LIN {X 261.750,Y 124.846,Z 181.546,A -154.500,B 90.000,C 0.000} C_DIS
LIN {X 261.491,Y 125.389,Z 179.119,A -154.382,B 90.000,C 0.000} C_DIS
LIN {X 261.280,Y 125.829,Z 176.668,A -154.285,B 90.000,C 0.000} C_DIS
LIN {X 261.097,Y 126.208,Z 174.203,A -154.202,B 90.000,C 0.000} C_DIS
LIN {X 261.001,Y 126.406,Z 172.680,A -154.159,B 90.000,C 0.000} C_DIS
LIN {X 260.699,Y 127.028,Z 175.082,A -154.022,B 90.000,C 0.000} C_DIS
LIN {X 260.678,Y 127.070,Z 175.258,A -154.013,B 90.000,C 0.000} C_DIS
LIN {X 260.668,Y 127.091,Z 175.443,A -154.008,B 90.000,C 0.000} C_DIS
LIN {X 260.648,Y 127.131,Z 175.543,A -153.999,B 90.000,C 0.000} C_DIS
LIN {X 260.511,Y 127.412,Z 176.567,A -153.938,B 90.000,C 0.000} C_DIS
LIN {X 260.496,Y 127.443,Z 176.806,A -153.931,B 90.000,C 0.000} C_DIS
LIN {X 260.198,Y 128.050,Z 179.115,A -153.797,B 90.000,C 0.000} C_DIS
LIN {X 260.188,Y 128.071,Z 179.244,A -153.792,B 90.000,C 0.000} C_DIS
LIN {X 260.152,Y 128.145,Z 179.466,A -153.776,B 90.000,C 0.000} C_DIS
LIN {X 260.141,Y 128.166,Z 179.594,A -153.772,B 90.000,C 0.000} C_DIS
LIN {X 259.890,Y 128.674,Z 181.403,A -153.660,B 90.000,C 0.000} C_DIS
LIN {X 259.860,Y 128.735,Z 181.801,A -153.646,B 90.000,C 0.000} C_DIS
LIN {X 259.844,Y 128.768,Z 181.915,A -153.639,B 90.000,C 0.000} C_DIS
LIN {X 259.830,Y 128.797,Z 181.972,A -153.633,B 90.000,C 0.000} C_DIS
LIN {X 259.824,Y 128.808,Z 182.029,A -153.630,B 90.000,C 0.000} C_DIS
LIN {X 259.588,Y 129.283,Z 183.707,A -153.525,B 90.000,C 0.000} C_DIS
LIN {X 259.577,Y 129.304,Z 183.864,A -153.521,B 90.000,C 0.000} C_DIS
LIN {X 259.564,Y 129.330,Z 183.963,A -153.515,B 90.000,C 0.000} C_DIS
LIN {X 259.518,Y 129.423,Z 184.177,A -153.494,B 90.000,C 0.000} C_DIS
LIN {X 259.392,Y 129.675,Z 185.123,A -153.439,B 90.000,C 0.000} C_DIS
LIN {X 259.382,Y 129.696,Z 185.286,A -153.434,B 90.000,C 0.000} C_DIS
LIN {X 259.358,Y 129.744,Z 185.386,A -153.423,B 90.000,C 0.000} C_DIS
LIN {X 259.343,Y 129.773,Z 185.423,A -153.417,B 90.000,C 0.000} C_DIS
LIN {X 259.334,Y 129.792,Z 185.531,A -153.413,B 90.000,C 0.000} C_DIS
LIN {X 259.124,Y 130.210,Z 186.922,A -153.320,B 90.000,C 0.000} C_DIS
LIN {X 258.879,Y 130.697,Z 188.742,A -153.213,B 90.000,C 0.000} C_DIS
LIN {X 258.539,Y 131.368,Z 190.848,A -153.064,B 90.000,C 0.000} C_DIS
LIN {X 258.522,Y 131.401,Z 191.075,A -153.057,B 90.000,C 0.000} C_DIS
LIN {X 258.356,Y 131.727,Z 191.986,A -152.985,B 90.000,C 0.000} C_DIS
LIN {X 258.326,Y 131.787,Z 192.346,A -152.971,B 90.000,C 0.000} C_DIS
LIN {X 258.310,Y 131.819,Z 192.384,A -152.964,B 90.000,C 0.000} C_DIS
LIN {X 258.290,Y 131.857,Z 192.498,A -152.956,B 90.000,C 0.000} C_DIS
LIN {X 258.283,Y 131.871,Z 192.611,A -152.952,B 90.000,C 0.000} C_DIS
LIN {X 258.179,Y 132.075,Z 193.180,A -152.907,B 90.000,C 0.000} C_DIS
LIN {X 258.171,Y 132.089,Z 193.294,A -152.904,B 90.000,C 0.000} C_DIS
LIN {X 258.154,Y 132.122,Z 193.408,A -152.897,B 90.000,C 0.000} C_DIS
LIN {X 258.140,Y 132.150,Z 193.465,A -152.891,B 90.000,C 0.000} C_DIS
LIN {X 258.134,Y 132.162,Z 193.522,A -152.888,B 90.000,C 0.000} C_DIS
LIN {X 257.980,Y 132.463,Z 194.356,A -152.821,B 90.000,C 0.000} C_DIS
LIN {X 257.975,Y 132.473,Z 194.455,A -152.819,B 90.000,C 0.000} C_DIS
LIN {X 257.839,Y 132.737,Z 195.229,A -152.760,B 90.000,C 0.000} C_DIS
LIN {X 257.834,Y 132.747,Z 195.342,A -152.758,B 90.000,C 0.000} C_DIS
LIN {X 257.799,Y 132.815,Z 195.542,A -152.743,B 90.000,C 0.000} C_DIS
LIN {X 257.793,Y 132.826,Z 195.627,A -152.741,B 90.000,C 0.000} C_DIS
LIN {X 257.655,Y 133.093,Z 196.400,A -152.681,B 90.000,C 0.000} C_DIS
LIN {X 257.650,Y 133.103,Z 196.500,A -152.679,B 90.000,C 0.000} C_DIS
LIN {X 257.529,Y 133.337,Z 197.076,A -152.627,B 90.000,C 0.000} C_DIS
LIN {X 257.435,Y 133.518,Z 197.632,A -152.587,B 90.000,C 0.000} C_DIS
LIN {X 257.056,Y 134.247,Z 199.808,A -152.424,B 90.000,C 0.000} C_DIS
LIN {X 256.932,Y 134.483,Z 200.387,A -152.372,B 90.000,C 0.000} C_DIS
LIN {X 256.928,Y 134.491,Z 200.486,A -152.370,B 90.000,C 0.000} C_DIS
LIN {X 256.816,Y 134.705,Z 201.032,A -152.322,B 90.000,C 0.000} C_DIS
LIN {X 256.810,Y 134.716,Z 201.146,A -152.320,B 90.000,C 0.000} C_DIS
LIN {X 256.793,Y 134.749,Z 201.260,A -152.312,B 90.000,C 0.000} C_DIS
LIN {X 256.778,Y 134.777,Z 201.316,A -152.306,B 90.000,C 0.000} C_DIS
LIN {X 256.417,Y 135.464,Z 203.137,A -152.153,B 90.000,C 0.000} C_DIS
LIN {X 256.396,Y 135.504,Z 203.251,A -152.144,B 90.000,C 0.000} C_DIS
LIN {X 256.367,Y 135.557,Z 203.338,A -152.132,B 90.000,C 0.000} C_DIS
LIN {X 256.288,Y 135.707,Z 203.870,A -152.098,B 90.000,C 0.000} C_DIS
LIN {X 256.269,Y 135.744,Z 203.927,A -152.090,B 90.000,C 0.000} C_DIS
LIN {X 256.128,Y 136.010,Z 204.533,A -152.031,B 90.000,C 0.000} C_DIS
LIN {X 256.051,Y 136.154,Z 205.052,A -151.998,B 90.000,C 0.000} C_DIS
LIN {X 256.028,Y 136.196,Z 205.122,A -151.989,B 90.000,C 0.000} C_DIS
LIN {X 255.803,Y 136.620,Z 206.186,A -151.894,B 90.000,C 0.000} C_DIS
LIN {X 255.794,Y 136.635,Z 206.270,A -151.891,B 90.000,C 0.000} C_DIS
LIN {X 255.561,Y 137.072,Z 207.291,A -151.793,B 90.000,C 0.000} C_DIS
LIN {X 255.543,Y 137.106,Z 207.333,A -151.785,B 90.000,C 0.000} C_DIS
LIN {X 255.484,Y 137.214,Z 207.749,A -151.761,B 90.000,C 0.000} C_DIS
LIN {X 255.456,Y 137.267,Z 207.803,A -151.749,B 90.000,C 0.000} C_DIS
LIN {X 255.434,Y 137.308,Z 207.916,A -151.740,B 90.000,C 0.000} C_DIS
LIN {X 255.235,Y 137.678,Z 208.850,A -151.657,B 90.000,C 0.000} C_DIS
LIN {X 255.220,Y 137.705,Z 208.884,A -151.651,B 90.000,C 0.000} C_DIS
LIN {X 255.172,Y 137.794,Z 209.086,A -151.631,B 90.000,C 0.000} C_DIS
LIN {X 254.804,Y 138.474,Z 210.647,A -151.478,B 90.000,C 0.000} C_DIS
LIN {X 254.783,Y 138.513,Z 210.761,A -151.469,B 90.000,C 0.000} C_DIS
LIN {X 254.754,Y 138.566,Z 210.842,A -151.457,B 90.000,C 0.000} C_DIS
LIN {X 254.706,Y 138.653,Z 211.023,A -151.438,B 90.000,C 0.000} C_DIS
LIN {X 254.662,Y 138.735,Z 211.155,A -151.419,B 90.000,C 0.000} C_DIS
LIN {X 254.427,Y 139.165,Z 212.216,A -151.322,B 90.000,C 0.000} C_DIS
LIN {X 254.398,Y 139.218,Z 212.297,A -151.311,B 90.000,C 0.000} C_DIS
LIN {X 254.374,Y 139.262,Z 212.411,A -151.301,B 90.000,C 0.000} C_DIS
LIN {X 254.345,Y 139.315,Z 212.492,A -151.289,B 90.000,C 0.000} C_DIS
LIN {X 254.303,Y 139.391,Z 212.661,A -151.271,B 90.000,C 0.000} C_DIS
LIN {X 254.263,Y 139.465,Z 212.780,A -151.255,B 90.000,C 0.000} C_DIS
LIN {X 254.224,Y 139.536,Z 212.973,A -151.239,B 90.000,C 0.000} C_DIS
LIN {X 254.200,Y 139.579,Z 213.172,A -151.229,B 90.000,C 0.000} C_DIS
LIN {X 253.989,Y 139.963,Z 213.976,A -151.143,B 90.000,C 0.000} C_DIS
LIN {X 253.943,Y 140.047,Z 214.108,A -151.124,B 90.000,C 0.000} C_DIS
LIN {X 253.906,Y 140.112,Z 214.264,A -151.109,B 90.000,C 0.000} C_DIS
LIN {X 253.792,Y 140.320,Z 214.630,A -151.062,B 90.000,C 0.000} C_DIS
LIN {X 253.771,Y 140.359,Z 214.744,A -151.053,B 90.000,C 0.000} C_DIS
LIN {X 253.712,Y 140.464,Z 214.915,A -151.030,B 90.000,C 0.000} C_DIS
LIN {X 253.688,Y 140.508,Z 215.028,A -151.020,B 90.000,C 0.000} C_DIS
LIN {X 253.659,Y 140.561,Z 215.105,A -151.008,B 90.000,C 0.000} C_DIS
LIN {X 253.548,Y 140.760,Z 215.521,A -150.963,B 90.000,C 0.000} C_DIS
LIN {X 253.519,Y 140.812,Z 215.597,A -150.951,B 90.000,C 0.000} C_DIS
LIN {X 253.495,Y 140.856,Z 215.711,A -150.941,B 90.000,C 0.000} C_DIS
LIN {X 253.436,Y 140.961,Z 215.882,A -150.917,B 90.000,C 0.000} C_DIS
LIN {X 253.412,Y 141.005,Z 215.996,A -150.907,B 90.000,C 0.000} C_DIS
LIN {X 253.382,Y 141.058,Z 216.072,A -150.895,B 90.000,C 0.000} C_DIS
LIN {X 253.143,Y 141.487,Z 216.805,A -150.798,B 90.000,C 0.000} C_DIS
LIN {X 252.855,Y 142.002,Z 217.779,A -150.682,B 90.000,C 0.000} C_DIS
LIN {X 252.797,Y 142.105,Z 217.992,A -150.658,B 90.000,C 0.000} C_DIS
LIN {X 252.693,Y 142.289,Z 218.286,A -150.616,B 90.000,C 0.000} C_DIS
LIN {X 252.624,Y 142.412,Z 218.442,A -150.589,B 90.000,C 0.000} C_DIS
LIN {X 252.618,Y 142.423,Z 218.499,A -150.586,B 90.000,C 0.000} C_DIS
LIN {X 252.605,Y 142.445,Z 218.556,A -150.581,B 90.000,C 0.000} C_DIS
LIN {X 252.529,Y 142.581,Z 218.764,A -150.550,B 90.000,C 0.000} C_DIS
LIN {X 252.408,Y 142.795,Z 219.122,A -150.502,B 90.000,C 0.000} C_DIS
LIN {X 252.378,Y 142.847,Z 219.182,A -150.490,B 90.000,C 0.000} C_DIS
LIN {X 252.353,Y 142.891,Z 219.296,A -150.480,B 90.000,C 0.000} C_DIS
LIN {X 252.291,Y 143.001,Z 219.466,A -150.455,B 90.000,C 0.000} C_DIS
LIN {X 252.274,Y 143.031,Z 219.499,A -150.448,B 90.000,C 0.000} C_DIS
LIN {X 251.761,Y 143.932,Z 220.886,A -150.243,B 90.000,C 0.000} C_DIS
LIN {X 251.728,Y 143.990,Z 220.946,A -150.230,B 90.000,C 0.000} C_DIS
LIN {X 251.713,Y 144.017,Z 220.981,A -150.224,B 90.000,C 0.000} C_DIS
LIN {X 251.654,Y 144.119,Z 221.173,A -150.201,B 90.000,C 0.000} C_DIS
LIN {X 250.995,Y 145.264,Z 222.709,A -149.940,B 90.000,C 0.000} C_DIS
LIN {X 250.952,Y 145.338,Z 222.766,A -149.923,B 90.000,C 0.000} C_DIS
LIN {X 250.867,Y 145.485,Z 222.937,A -149.889,B 90.000,C 0.000} C_DIS
LIN {X 250.824,Y 145.559,Z 222.982,A -149.872,B 90.000,C 0.000} C_DIS
LIN {X 250.161,Y 146.696,Z 224.246,A -149.612,B 90.000,C 0.000} C_DIS
LIN {X 249.905,Y 147.131,Z 224.706,A -149.513,B 90.000,C 0.000} C_DIS
LIN {X 249.753,Y 147.388,Z 224.928,A -149.454,B 90.000,C 0.000} C_DIS
LIN {X 248.658,Y 149.229,Z 226.216,A -149.030,B 90.000,C 0.000} C_DIS
LIN {X 248.413,Y 149.636,Z 226.445,A -148.937,B 90.000,C 0.000} C_DIS
LIN {X 248.308,Y 149.810,Z 226.460,A -148.897,B 90.000,C 0.000} C_DIS
LIN {X 248.170,Y 150.038,Z 226.328,A -148.844,B 90.000,C 0.000} C_DIS
LIN {X 247.772,Y 150.695,Z 225.771,A -148.692,B 90.000,C 0.000} C_DIS
LIN {X 247.484,Y 151.167,Z 225.386,A -148.583,B 90.000,C 0.000} C_DIS
LIN {X 247.345,Y 151.395,Z 225.255,A -148.530,B 90.000,C 0.000} C_DIS
LIN {X 247.299,Y 151.470,Z 225.156,A -148.513,B 90.000,C 0.000} C_DIS
LIN {X 246.570,Y 152.654,Z 224.116,A -148.238,B 90.000,C 0.000} C_DIS
LIN {X 246.521,Y 152.734,Z 224.018,A -148.219,B 90.000,C 0.000} C_DIS
LIN {X 246.069,Y 153.460,Z 223.362,A -148.051,B 90.000,C 0.000} C_DIS
LIN {X 245.953,Y 153.646,Z 223.134,A -148.007,B 90.000,C 0.000} C_DIS
LIN {X 244.939,Y 155.258,Z 221.514,A -147.631,B 90.000,C 0.000} C_DIS
LIN {X 244.768,Y 155.527,Z 221.240,A -147.568,B 90.000,C 0.000} C_DIS
LIN {X 244.507,Y 155.937,Z 220.768,A -147.472,B 90.000,C 0.000} C_DIS
LIN {X 244.472,Y 155.992,Z 220.682,A -147.459,B 90.000,C 0.000} C_DIS
LIN {X 244.123,Y 156.537,Z 220.149,A -147.331,B 90.000,C 0.000} C_DIS
LIN {X 244.079,Y 156.606,Z 220.034,A -147.315,B 90.000,C 0.000} C_DIS
LIN {X 243.939,Y 156.824,Z 219.782,A -147.264,B 90.000,C 0.000} C_DIS
LIN {X 243.910,Y 156.869,Z 219.759,A -147.253,B 90.000,C 0.000} C_DIS
LIN {X 243.416,Y 157.634,Z 218.840,A -147.073,B 90.000,C 0.000} C_DIS
LIN {X 243.386,Y 157.681,Z 218.755,A -147.062,B 90.000,C 0.000} C_DIS
LIN {X 243.293,Y 157.825,Z 218.583,A -147.028,B 90.000,C 0.000} C_DIS
LIN {X 243.200,Y 157.968,Z 218.351,A -146.995,B 90.000,C 0.000} C_DIS
LIN {X 243.107,Y 158.111,Z 218.186,A -146.961,B 90.000,C 0.000} C_DIS
LIN {X 242.920,Y 158.397,Z 217.804,A -146.894,B 90.000,C 0.000} C_DIS
LIN {X 242.889,Y 158.445,Z 217.788,A -146.882,B 90.000,C 0.000} C_DIS
LIN {X 242.858,Y 158.492,Z 217.763,A -146.871,B 90.000,C 0.000} C_DIS
LIN {X 242.392,Y 159.204,Z 216.749,A -146.703,B 90.000,C 0.000} C_DIS
LIN {X 242.344,Y 159.278,Z 216.678,A -146.686,B 90.000,C 0.000} C_DIS
LIN {X 242.297,Y 159.349,Z 216.591,A -146.669,B 90.000,C 0.000} C_DIS
LIN {X 242.250,Y 159.420,Z 216.471,A -146.652,B 90.000,C 0.000} C_DIS
LIN {X 242.203,Y 159.492,Z 216.388,A -146.635,B 90.000,C 0.000} C_DIS
LIN {X 242.148,Y 159.575,Z 216.229,A -146.615,B 90.000,C 0.000} C_DIS
LIN {X 241.701,Y 160.251,Z 215.249,A -146.455,B 90.000,C 0.000} C_DIS
LIN {X 241.639,Y 160.346,Z 215.211,A -146.433,B 90.000,C 0.000} C_DIS
LIN {X 241.513,Y 160.536,Z 214.821,A -146.388,B 90.000,C 0.000} C_DIS
LIN {X 241.418,Y 160.678,Z 214.665,A -146.354,B 90.000,C 0.000} C_DIS
LIN {X 241.323,Y 160.820,Z 214.461,A -146.320,B 90.000,C 0.000} C_DIS
LIN {X 241.136,Y 161.101,Z 213.937,A -146.253,B 90.000,C 0.000} C_DIS
LIN {X 242.353,Y 159.265,Z 212.755,A -146.689,B 90.000,C 0.000} C_DIS
LIN {X 243.523,Y 157.470,Z 211.467,A -147.112,B 90.000,C 0.000} C_DIS
LIN {X 244.293,Y 156.271,Z 210.534,A -147.393,B 90.000,C 0.000} C_DIS
LIN {X 245.035,Y 155.106,Z 209.566,A -147.666,B 90.000,C 0.000} C_DIS
LIN {X 245.147,Y 154.928,Z 209.396,A -147.708,B 90.000,C 0.000} C_DIS
LIN {X 245.353,Y 154.603,Z 209.168,A -147.784,B 90.000,C 0.000} C_DIS
LIN {X 245.362,Y 154.588,Z 209.113,A -147.787,B 90.000,C 0.000} C_DIS
LIN {X 245.421,Y 154.495,Z 209.021,A -147.809,B 90.000,C 0.000} C_DIS
LIN {X 245.498,Y 154.372,Z 208.933,A -147.838,B 90.000,C 0.000} C_DIS
LIN {X 245.548,Y 154.292,Z 208.843,A -147.857,B 90.000,C 0.000} C_DIS
LIN {X 245.868,Y 153.781,Z 208.428,A -147.976,B 90.000,C 0.000} C_DIS
LIN {X 245.876,Y 153.770,Z 208.372,A -147.978,B 90.000,C 0.000} C_DIS
LIN {X 245.905,Y 153.723,Z 208.315,A -147.989,B 90.000,C 0.000} C_DIS
LIN {X 246.345,Y 153.017,Z 207.660,A -148.153,B 90.000,C 0.000} C_DIS
LIN {X 246.421,Y 152.894,Z 207.575,A -148.182,B 90.000,C 0.000} C_DIS
LIN {X 246.750,Y 152.363,Z 207.063,A -148.305,B 90.000,C 0.000} C_DIS
LIN {X 246.791,Y 152.296,Z 206.978,A -148.321,B 90.000,C 0.000} C_DIS
LIN {X 246.820,Y 152.250,Z 206.892,A -148.332,B 90.000,C 0.000} C_DIS
LIN {X 247.039,Y 151.894,Z 206.586,A -148.414,B 90.000,C 0.000} C_DIS
LIN {X 247.052,Y 151.872,Z 206.551,A -148.419,B 90.000,C 0.000} C_DIS
LIN {X 247.541,Y 151.074,Z 205.811,A -148.604,B 90.000,C 0.000} C_DIS
LIN {X 247.561,Y 151.041,Z 205.697,A -148.612,B 90.000,C 0.000} C_DIS
LIN {X 247.837,Y 150.588,Z 205.299,A -148.717,B 90.000,C 0.000} C_DIS
LIN {X 247.846,Y 150.573,Z 205.242,A -148.720,B 90.000,C 0.000} C_DIS
LIN {X 247.868,Y 150.537,Z 205.185,A -148.728,B 90.000,C 0.000} C_DIS
LIN {X 248.834,Y 148.936,Z 203.527,A -149.098,B 90.000,C 0.000} C_DIS
LIN {X 248.863,Y 148.886,Z 203.478,A -149.109,B 90.000,C 0.000} C_DIS
LIN {X 248.888,Y 148.844,Z 203.365,A -149.119,B 90.000,C 0.000} C_DIS
LIN {X 249.802,Y 147.305,Z 201.620,A -149.473,B 90.000,C 0.000} C_DIS
LIN {X 250.670,Y 145.824,Z 199.802,A -149.812,B 90.000,C 0.000} C_DIS
LIN {X 250.709,Y 145.756,Z 199.719,A -149.827,B 90.000,C 0.000} C_DIS
LIN {X 250.795,Y 145.608,Z 199.609,A -149.861,B 90.000,C 0.000} C_DIS
LIN {X 251.434,Y 144.502,Z 198.183,A -150.114,B 90.000,C 0.000} C_DIS
LIN {X 251.448,Y 144.478,Z 198.130,A -150.119,B 90.000,C 0.000} C_DIS
LIN {X 251.478,Y 144.426,Z 198.045,A -150.131,B 90.000,C 0.000} C_DIS
LIN {X 251.521,Y 144.352,Z 197.960,A -150.148,B 90.000,C 0.000} C_DIS
LIN {X 251.563,Y 144.278,Z 197.895,A -150.165,B 90.000,C 0.000} C_DIS
LIN {X 251.761,Y 143.932,Z 197.394,A -150.243,B 90.000,C 0.000} C_DIS
LIN {X 251.803,Y 143.858,Z 197.334,A -150.260,B 90.000,C 0.000} C_DIS
LIN {X 251.846,Y 143.784,Z 197.248,A -150.277,B 90.000,C 0.000} C_DIS
LIN {X 251.875,Y 143.732,Z 197.163,A -150.289,B 90.000,C 0.000} C_DIS
LIN {X 251.889,Y 143.708,Z 197.110,A -150.294,B 90.000,C 0.000} C_DIS
LIN {X 251.932,Y 143.633,Z 197.020,A -150.311,B 90.000,C 0.000} C_DIS
LIN {X 251.976,Y 143.555,Z 196.952,A -150.329,B 90.000,C 0.000} C_DIS
LIN {X 252.193,Y 143.174,Z 196.348,A -150.416,B 90.000,C 0.000} C_DIS
LIN {X 252.238,Y 143.095,Z 196.282,A -150.434,B 90.000,C 0.000} C_DIS
LIN {X 252.280,Y 143.020,Z 196.192,A -150.451,B 90.000,C 0.000} C_DIS
LIN {X 252.294,Y 142.995,Z 196.139,A -150.456,B 90.000,C 0.000} C_DIS
LIN {X 252.324,Y 142.943,Z 196.054,A -150.468,B 90.000,C 0.000} C_DIS
LIN {X 252.366,Y 142.869,Z 195.968,A -150.485,B 90.000,C 0.000} C_DIS
LIN {X 252.408,Y 142.795,Z 195.907,A -150.502,B 90.000,C 0.000} C_DIS
LIN {X 252.833,Y 142.040,Z 194.805,A -150.673,B 90.000,C 0.000} C_DIS
LIN {X 252.883,Y 141.952,Z 194.714,A -150.693,B 90.000,C 0.000} C_DIS
LIN {X 253.244,Y 141.306,Z 193.754,A -150.839,B 90.000,C 0.000} C_DIS
LIN {X 253.292,Y 141.221,Z 193.658,A -150.859,B 90.000,C 0.000} C_DIS
LIN {X 253.336,Y 141.141,Z 193.501,A -150.877,B 90.000,C 0.000} C_DIS
LIN {X 253.796,Y 140.312,Z 192.272,A -151.064,B 90.000,C 0.000} C_DIS
LIN {X 253.845,Y 140.223,Z 192.182,A -151.084,B 90.000,C 0.000} C_DIS
LIN {X 254.455,Y 139.113,Z 190.433,A -151.334,B 90.000,C 0.000} C_DIS
LIN {X 255.150,Y 137.834,Z 188.401,A -151.622,B 90.000,C 0.000} C_DIS
LIN {X 255.460,Y 137.260,Z 187.428,A -151.751,B 90.000,C 0.000} C_DIS
LIN {X 255.560,Y 137.074,Z 187.135,A -151.792,B 90.000,C 0.000} C_DIS
LIN {X 255.626,Y 136.950,Z 186.979,A -151.820,B 90.000,C 0.000} C_DIS
LIN {X 255.641,Y 136.922,Z 186.865,A -151.826,B 90.000,C 0.000} C_DIS
LIN {X 255.798,Y 136.628,Z 186.373,A -151.892,B 90.000,C 0.000} C_DIS
LIN {X 256.050,Y 136.157,Z 185.556,A -151.998,B 90.000,C 0.000} C_DIS
LIN {X 256.073,Y 136.113,Z 185.442,A -152.008,B 90.000,C 0.000} C_DIS
LIN {X 256.129,Y 136.007,Z 185.272,A -152.031,B 90.000,C 0.000} C_DIS
LIN {X 256.153,Y 135.962,Z 185.158,A -152.041,B 90.000,C 0.000} C_DIS
LIN {X 256.181,Y 135.909,Z 185.081,A -152.053,B 90.000,C 0.000} C_DIS
LIN {X 256.477,Y 135.350,Z 184.134,A -152.178,B 90.000,C 0.000} C_DIS
LIN {X 256.561,Y 135.191,Z 183.770,A -152.214,B 90.000,C 0.000} C_DIS
LIN {X 256.606,Y 135.104,Z 183.654,A -152.233,B 90.000,C 0.000} C_DIS
LIN {X 256.697,Y 134.931,Z 183.292,A -152.272,B 90.000,C 0.000} C_DIS
LIN {X 256.806,Y 134.725,Z 182.917,A -152.318,B 90.000,C 0.000} C_DIS
LIN {X 256.843,Y 134.654,Z 182.813,A -152.334,B 90.000,C 0.000} C_DIS
LIN {X 256.928,Y 134.492,Z 182.484,A -152.370,B 90.000,C 0.000} C_DIS
LIN {X 256.950,Y 134.449,Z 182.423,A -152.379,B 90.000,C 0.000} C_DIS
LIN {X 257.266,Y 133.844,Z 181.127,A -152.514,B 90.000,C 0.000} C_DIS
LIN {X 257.333,Y 133.715,Z 180.936,A -152.543,B 90.000,C 0.000} C_DIS
LIN {X 257.423,Y 133.541,Z 180.574,A -152.581,B 90.000,C 0.000} C_DIS
LIN {X 257.451,Y 133.488,Z 180.493,A -152.593,B 90.000,C 0.000} C_DIS
LIN {X 257.474,Y 133.443,Z 180.379,A -152.603,B 90.000,C 0.000} C_DIS
LIN {X 257.502,Y 133.390,Z 180.302,A -152.615,B 90.000,C 0.000} C_DIS
LIN {X 257.606,Y 133.188,Z 179.886,A -152.660,B 90.000,C 0.000} C_DIS
LIN {X 257.634,Y 133.134,Z 179.810,A -152.672,B 90.000,C 0.000} C_DIS
LIN {X 257.647,Y 133.109,Z 179.758,A -152.678,B 90.000,C 0.000} C_DIS
LIN {X 257.652,Y 133.099,Z 179.687,A -152.680,B 90.000,C 0.000} C_DIS
LIN {X 257.848,Y 132.720,Z 178.966,A -152.764,B 90.000,C 0.000} C_DIS
LIN {X 257.932,Y 132.556,Z 178.501,A -152.801,B 90.000,C 0.000} C_DIS
LIN {X 257.997,Y 132.429,Z 178.241,A -152.829,B 90.000,C 0.000} C_DIS
LIN {X 258.025,Y 132.375,Z 178.160,A -152.841,B 90.000,C 0.000} C_DIS
LIN {X 258.048,Y 132.331,Z 178.046,A -152.851,B 90.000,C 0.000} C_DIS
LIN {X 258.075,Y 132.277,Z 177.965,A -152.862,B 90.000,C 0.000} C_DIS
LIN {X 258.386,Y 131.669,Z 176.591,A -152.997,B 90.000,C 0.000} C_DIS
LIN {X 258.413,Y 131.615,Z 176.510,A -153.009,B 90.000,C 0.000} C_DIS
LIN {X 258.433,Y 131.577,Z 176.396,A -153.018,B 90.000,C 0.000} C_DIS
LIN {X 258.911,Y 130.633,Z 174.131,A -153.227,B 90.000,C 0.000} C_DIS
LIN {X 258.969,Y 130.518,Z 173.878,A -153.252,B 90.000,C 0.000} C_DIS
LIN {X 259.259,Y 129.942,Z 172.129,A -153.380,B 90.000,C 0.000} C_DIS
LIN {X 259.266,Y 129.928,Z 172.015,A -153.383,B 90.000,C 0.000} C_DIS
LIN {X 259.353,Y 129.754,Z 171.389,A -153.421,B 90.000,C 0.000} C_DIS
LIN {X 259.360,Y 129.740,Z 171.275,A -153.424,B 90.000,C 0.000} C_DIS
LIN {X 259.393,Y 129.674,Z 171.119,A -153.439,B 90.000,C 0.000} C_DIS
LIN {X 259.671,Y 129.116,Z 168.698,A -153.562,B 90.000,C 0.000} C_DIS
LIN {X 259.684,Y 129.090,Z 168.587,A -153.568,B 90.000,C 0.000} C_DIS
LIN {X 259.716,Y 129.025,Z 168.431,A -153.582,B 90.000,C 0.000} C_DIS
LIN {X 259.723,Y 129.011,Z 168.317,A -153.585,B 90.000,C 0.000} C_DIS
LIN {X 259.842,Y 128.773,Z 167.322,A -153.638,B 90.000,C 0.000} C_DIS
LIN {X 259.854,Y 128.748,Z 167.232,A -153.643,B 90.000,C 0.000} C_DIS
LIN {X 259.890,Y 128.674,Z 167.079,A -153.660,B 90.000,C 0.000} C_DIS
LIN {X 259.901,Y 128.653,Z 166.894,A -153.664,B 90.000,C 0.000} C_DIS
LIN {X 260.187,Y 128.072,Z 164.480,A -153.792,B 90.000,C 0.000} C_DIS
LIN {X 260.196,Y 128.054,Z 164.405,A -153.796,B 90.000,C 0.000} C_DIS
LIN {X 258.402,Y 127.171,Z 164.405,A -153.796,B 90.000,C 0.000} C_DIS
WAIT SEC 0.1
RET=EKI_SetBool("oxy","torchState",FALSE)
RET = EKI_Send("oxy","torchState")
LIN {X 242.252,Y 119.223,Z 164.405,A -153.796,B 90.000,C 0.000} C_DIS
LIN {X 245.422,Y 112.552,Z 164.348,A -155.364,B 90.000,C 0.000} C_DIS
LIN {X 261.784,Y 120.055,Z 164.348,A -155.364,B 90.000,C 0.000} C_DIS
LIN {X 263.602,Y 120.889,Z 164.348,A -155.364,B 90.000,C 0.000} C_DIS
WAIT SEC 1
RET=EKI_SetBool("oxy","torchState",TRUE)
RET = EKI_Send("oxy","torchState")
LIN {X 263.563,Y 120.973,Z 165.813,A -155.345,B 90.000,C 0.000} C_DIS
LIN {X 263.565,Y 120.969,Z 166.657,A -155.346,B 90.000,C 0.000} C_DIS
LIN {X 263.556,Y 120.989,Z 166.730,A -155.342,B 90.000,C 0.000} C_DIS
LIN {X 263.645,Y 120.795,Z 169.220,A -155.384,B 90.000,C 0.000} C_DIS
LIN {X 263.775,Y 120.510,Z 170.942,A -155.446,B 90.000,C 0.000} C_DIS
LIN {X 264.136,Y 119.717,Z 173.285,A -155.618,B 90.000,C 0.000} C_DIS
LIN {X 264.561,Y 118.775,Z 175.562,A -155.822,B 90.000,C 0.000} C_DIS
LIN {X 264.902,Y 118.011,Z 177.202,A -155.988,B 90.000,C 0.000} C_DIS
LIN {X 265.110,Y 117.545,Z 178.103,A -156.088,B 90.000,C 0.000} C_DIS
LIN {X 265.524,Y 116.607,Z 179.841,A -156.291,B 90.000,C 0.000} C_DIS
LIN {X 265.592,Y 116.450,Z 180.055,A -156.325,B 90.000,C 0.000} C_DIS
LIN {X 265.684,Y 116.242,Z 180.473,A -156.370,B 90.000,C 0.000} C_DIS
LIN {X 265.834,Y 115.897,Z 180.982,A -156.444,B 90.000,C 0.000} C_DIS
LIN {X 265.886,Y 115.778,Z 181.234,A -156.470,B 90.000,C 0.000} C_DIS
LIN {X 266.457,Y 114.457,Z 183.278,A -156.754,B 90.000,C 0.000} C_DIS
LIN {X 266.607,Y 114.108,Z 183.792,A -156.829,B 90.000,C 0.000} C_DIS
LIN {X 266.783,Y 113.695,Z 184.351,A -156.918,B 90.000,C 0.000} C_DIS
LIN {X 266.811,Y 113.630,Z 184.483,A -156.932,B 90.000,C 0.000} C_DIS
LIN {X 266.856,Y 113.525,Z 184.520,A -156.954,B 90.000,C 0.000} C_DIS
LIN {X 266.945,Y 113.316,Z 184.911,A -156.999,B 90.000,C 0.000} C_DIS
LIN {X 267.011,Y 113.159,Z 185.073,A -157.033,B 90.000,C 0.000} C_DIS
LIN {X 267.034,Y 113.105,Z 185.158,A -157.045,B 90.000,C 0.000} C_DIS
LIN {X 267.071,Y 113.017,Z 185.253,A -157.063,B 90.000,C 0.000} C_DIS
LIN {X 267.121,Y 112.901,Z 185.449,A -157.088,B 90.000,C 0.000} C_DIS
LIN {X 267.564,Y 111.845,Z 186.835,A -157.314,B 90.000,C 0.000} C_DIS
LIN {X 267.695,Y 111.533,Z 187.250,A -157.381,B 90.000,C 0.000} C_DIS
LIN {X 267.717,Y 111.480,Z 187.292,A -157.393,B 90.000,C 0.000} C_DIS
LIN {X 267.738,Y 111.428,Z 187.309,A -157.404,B 90.000,C 0.000} C_DIS
LIN {X 267.891,Y 111.060,Z 187.840,A -157.483,B 90.000,C 0.000} C_DIS
LIN {X 267.935,Y 110.955,Z 187.882,A -157.505,B 90.000,C 0.000} C_DIS
LIN {X 268.087,Y 110.587,Z 188.412,A -157.584,B 90.000,C 0.000} C_DIS
LIN {X 268.109,Y 110.534,Z 188.430,A -157.595,B 90.000,C 0.000} C_DIS
LIN {X 268.130,Y 110.481,Z 188.454,A -157.606,B 90.000,C 0.000} C_DIS
LIN {X 268.583,Y 109.376,Z 189.820,A -157.842,B 90.000,C 0.000} C_DIS
LIN {X 268.603,Y 109.327,Z 189.854,A -157.853,B 90.000,C 0.000} C_DIS
LIN {X 268.637,Y 109.243,Z 189.941,A -157.871,B 90.000,C 0.000} C_DIS
LIN {X 268.661,Y 109.185,Z 190.035,A -157.883,B 90.000,C 0.000} C_DIS
LIN {X 269.243,Y 107.740,Z 191.588,A -158.191,B 90.000,C 0.000} C_DIS
LIN {X 269.266,Y 107.684,Z 191.613,A -158.203,B 90.000,C 0.000} C_DIS
LIN {X 269.300,Y 107.599,Z 191.695,A -158.221,B 90.000,C 0.000} C_DIS
LIN {X 269.328,Y 107.528,Z 191.786,A -158.236,B 90.000,C 0.000} C_DIS
LIN {X 269.357,Y 107.455,Z 191.847,A -158.251,B 90.000,C 0.000} C_DIS
LIN {X 269.412,Y 107.317,Z 191.934,A -158.281,B 90.000,C 0.000} C_DIS
LIN {X 269.566,Y 106.932,Z 192.348,A -158.363,B 90.000,C 0.000} C_DIS
LIN {X 269.620,Y 106.793,Z 192.554,A -158.392,B 90.000,C 0.000} C_DIS
LIN {X 269.842,Y 106.233,Z 193.043,A -158.511,B 90.000,C 0.000} C_DIS
LIN {X 269.894,Y 106.101,Z 193.255,A -158.539,B 90.000,C 0.000} C_DIS
LIN {X 270.373,Y 104.874,Z 194.375,A -158.799,B 90.000,C 0.000} C_DIS
LIN {X 270.390,Y 104.829,Z 194.435,A -158.809,B 90.000,C 0.000} C_DIS
LIN {X 270.409,Y 104.779,Z 194.463,A -158.819,B 90.000,C 0.000} C_DIS
LIN {X 270.442,Y 104.695,Z 194.549,A -158.837,B 90.000,C 0.000} C_DIS
LIN {X 270.467,Y 104.632,Z 194.638,A -158.851,B 90.000,C 0.000} C_DIS
LIN {X 270.535,Y 104.454,Z 194.762,A -158.888,B 90.000,C 0.000} C_DIS
LIN {X 270.745,Y 103.910,Z 195.249,A -159.004,B 90.000,C 0.000} C_DIS
LIN {X 270.769,Y 103.848,Z 195.339,A -159.017,B 90.000,C 0.000} C_DIS
LIN {X 270.801,Y 103.763,Z 195.425,A -159.035,B 90.000,C 0.000} C_DIS
LIN {X 270.820,Y 103.714,Z 195.453,A -159.045,B 90.000,C 0.000} C_DIS
LIN {X 270.840,Y 103.661,Z 195.513,A -159.056,B 90.000,C 0.000} C_DIS
LIN {X 271.527,Y 101.849,Z 197.093,A -159.439,B 90.000,C 0.000} C_DIS
LIN {X 271.664,Y 101.483,Z 197.391,A -159.516,B 90.000,C 0.000} C_DIS
LIN {X 271.685,Y 101.425,Z 197.451,A -159.528,B 90.000,C 0.000} C_DIS
LIN {X 271.704,Y 101.376,Z 197.479,A -159.539,B 90.000,C 0.000} C_DIS
LIN {X 271.766,Y 101.208,Z 197.644,A -159.574,B 90.000,C 0.000} C_DIS
LIN {X 271.785,Y 101.159,Z 197.663,A -159.585,B 90.000,C 0.000} C_DIS
LIN {X 272.177,Y 100.099,Z 198.529,A -159.808,B 90.000,C 0.000} C_DIS
LIN {X 272.199,Y 100.038,Z 198.595,A -159.821,B 90.000,C 0.000} C_DIS
LIN {X 272.212,Y 100.003,Z 198.624,A -159.828,B 90.000,C 0.000} C_DIS
LIN {X 272.335,Y 99.667,Z 198.870,A -159.899,B 90.000,C 0.000} C_DIS
LIN {X 272.356,Y 99.611,Z 198.936,A -159.911,B 90.000,C 0.000} C_DIS
LIN {X 272.369,Y 99.576,Z 198.966,A -159.918,B 90.000,C 0.000} C_DIS
LIN {X 273.063,Y 97.656,Z 200.406,A -160.321,B 90.000,C 0.000} C_DIS
LIN {X 273.091,Y 97.578,Z 200.466,A -160.338,B 90.000,C 0.000} C_DIS
LIN {X 273.129,Y 97.470,Z 200.517,A -160.360,B 90.000,C 0.000} C_DIS
LIN {X 273.149,Y 97.414,Z 200.577,A -160.372,B 90.000,C 0.000} C_DIS
LIN {X 273.269,Y 97.076,Z 200.822,A -160.443,B 90.000,C 0.000} C_DIS
LIN {X 273.339,Y 96.881,Z 200.978,A -160.484,B 90.000,C 0.000} C_DIS
LIN {X 273.358,Y 96.827,Z 201.004,A -160.495,B 90.000,C 0.000} C_DIS
LIN {X 273.377,Y 96.773,Z 201.018,A -160.506,B 90.000,C 0.000} C_DIS
LIN {X 273.528,Y 96.344,Z 201.376,A -160.596,B 90.000,C 0.000} C_DIS
LIN {X 273.665,Y 95.955,Z 201.633,A -160.678,B 90.000,C 0.000} C_DIS
LIN {X 273.717,Y 95.807,Z 201.713,A -160.709,B 90.000,C 0.000} C_DIS
LIN {X 273.904,Y 95.270,Z 202.118,A -160.821,B 90.000,C 0.000} C_DIS
LIN {X 273.932,Y 95.190,Z 202.170,A -160.838,B 90.000,C 0.000} C_DIS
LIN {X 273.972,Y 95.076,Z 202.268,A -160.862,B 90.000,C 0.000} C_DIS
LIN {X 274.091,Y 94.733,Z 202.447,A -160.934,B 90.000,C 0.000} C_DIS
LIN {X 274.133,Y 94.612,Z 202.544,A -160.959,B 90.000,C 0.000} C_DIS
LIN {X 274.818,Y 92.601,Z 203.862,A -161.379,B 90.000,C 0.000} C_DIS
LIN {X 274.942,Y 92.234,Z 204.078,A -161.455,B 90.000,C 0.000} C_DIS
LIN {X 274.979,Y 92.122,Z 204.162,A -161.478,B 90.000,C 0.000} C_DIS
LIN {X 275.097,Y 91.770,Z 204.305,A -161.552,B 90.000,C 0.000} C_DIS
LIN {X 275.134,Y 91.660,Z 204.391,A -161.575,B 90.000,C 0.000} C_DIS
LIN {X 275.205,Y 91.446,Z 204.495,A -161.619,B 90.000,C 0.000} C_DIS
LIN {X 275.625,Y 90.172,Z 205.242,A -161.884,B 90.000,C 0.000} C_DIS
LIN {X 275.650,Y 90.095,Z 205.303,A -161.900,B 90.000,C 0.000} C_DIS
LIN {X 275.668,Y 90.041,Z 205.328,A -161.912,B 90.000,C 0.000} C_DIS
LIN {X 275.685,Y 89.987,Z 205.341,A -161.923,B 90.000,C 0.000} C_DIS
LIN {X 275.824,Y 89.560,Z 205.531,A -162.011,B 90.000,C 0.000} C_DIS
LIN {X 276.068,Y 88.805,Z 205.996,A -162.168,B 90.000,C 0.000} C_DIS
LIN {X 276.090,Y 88.737,Z 206.007,A -162.182,B 90.000,C 0.000} C_DIS
LIN {X 276.262,Y 88.200,Z 206.259,A -162.294,B 90.000,C 0.000} C_DIS
LIN {X 276.555,Y 87.278,Z 206.726,A -162.485,B 90.000,C 0.000} C_DIS
LIN {X 276.593,Y 87.156,Z 206.747,A -162.510,B 90.000,C 0.000} C_DIS
LIN {X 276.623,Y 87.061,Z 206.774,A -162.530,B 90.000,C 0.000} C_DIS
LIN {X 276.787,Y 86.540,Z 207.016,A -162.638,B 90.000,C 0.000} C_DIS
LIN {X 276.816,Y 86.445,Z 207.025,A -162.657,B 90.000,C 0.000} C_DIS
LIN {X 277.064,Y 85.649,Z 207.363,A -162.822,B 90.000,C 0.000} C_DIS
LIN {X 277.080,Y 85.594,Z 207.376,A -162.833,B 90.000,C 0.000} C_DIS
LIN {X 277.127,Y 85.445,Z 207.452,A -162.864,B 90.000,C 0.000} C_DIS
LIN {X 277.178,Y 85.278,Z 207.483,A -162.899,B 90.000,C 0.000} C_DIS
LIN {X 277.229,Y 85.111,Z 207.423,A -162.933,B 90.000,C 0.000} C_DIS
LIN {X 277.265,Y 84.996,Z 207.256,A -162.957,B 90.000,C 0.000} C_DIS
LIN {X 277.464,Y 84.343,Z 205.986,A -163.092,B 90.000,C 0.000} C_DIS
LIN {X 277.480,Y 84.290,Z 205.925,A -163.103,B 90.000,C 0.000} C_DIS
LIN {X 277.533,Y 84.116,Z 205.641,A -163.139,B 90.000,C 0.000} C_DIS
LIN {X 277.546,Y 84.074,Z 205.527,A -163.147,B 90.000,C 0.000} C_DIS
LIN {X 277.563,Y 84.017,Z 205.438,A -163.159,B 90.000,C 0.000} C_DIS
LIN {X 277.650,Y 83.730,Z 204.853,A -163.218,B 90.000,C 0.000} C_DIS
LIN {X 277.653,Y 83.720,Z 204.782,A -163.221,B 90.000,C 0.000} C_DIS
LIN {X 277.661,Y 83.693,Z 204.730,A -163.226,B 90.000,C 0.000} C_DIS
LIN {X 277.678,Y 83.635,Z 204.649,A -163.238,B 90.000,C 0.000} C_DIS
LIN {X 277.699,Y 83.567,Z 204.490,A -163.252,B 90.000,C 0.000} C_DIS
LIN {X 277.890,Y 82.930,Z 203.163,A -163.383,B 90.000,C 0.000} C_DIS
LIN {X 277.914,Y 82.847,Z 203.046,A -163.401,B 90.000,C 0.000} C_DIS
LIN {X 277.939,Y 82.763,Z 202.877,A -163.418,B 90.000,C 0.000} C_DIS
LIN {X 277.956,Y 82.705,Z 202.796,A -163.430,B 90.000,C 0.000} C_DIS
LIN {X 277.971,Y 82.657,Z 202.682,A -163.440,B 90.000,C 0.000} C_DIS
LIN {X 278.004,Y 82.545,Z 202.511,A -163.463,B 90.000,C 0.000} C_DIS
LIN {X 278.018,Y 82.500,Z 202.469,A -163.472,B 90.000,C 0.000} C_DIS
LIN {X 278.309,Y 81.512,Z 200.191,A -163.675,B 90.000,C 0.000} C_DIS
LIN {X 278.345,Y 81.390,Z 199.951,A -163.701,B 90.000,C 0.000} C_DIS
LIN {X 278.354,Y 81.359,Z 199.837,A -163.707,B 90.000,C 0.000} C_DIS
LIN {X 278.491,Y 80.886,Z 198.861,A -163.804,B 90.000,C 0.000} C_DIS
LIN {X 278.502,Y 80.851,Z 198.642,A -163.812,B 90.000,C 0.000} C_DIS
LIN {X 278.517,Y 80.798,Z 198.561,A -163.822,B 90.000,C 0.000} C_DIS
LIN {X 278.556,Y 80.664,Z 198.301,A -163.850,B 90.000,C 0.000} C_DIS
LIN {X 278.560,Y 80.651,Z 198.230,A -163.853,B 90.000,C 0.000} C_DIS
LIN {X 278.770,Y 79.921,Z 196.480,A -164.003,B 90.000,C 0.000} C_DIS
LIN {X 278.784,Y 79.873,Z 196.253,A -164.013,B 90.000,C 0.000} C_DIS
LIN {X 278.942,Y 79.317,Z 194.887,A -164.127,B 90.000,C 0.000} C_DIS
LIN {X 278.955,Y 79.271,Z 194.660,A -164.136,B 90.000,C 0.000} C_DIS
LIN {X 279.132,Y 78.647,Z 193.058,A -164.264,B 90.000,C 0.000} C_DIS
LIN {X 279.141,Y 78.614,Z 192.839,A -164.271,B 90.000,C 0.000} C_DIS
LIN {X 279.203,Y 78.394,Z 192.270,A -164.316,B 90.000,C 0.000} C_DIS
LIN {X 279.216,Y 78.348,Z 192.199,A -164.326,B 90.000,C 0.000} C_DIS
LIN {X 279.328,Y 77.949,Z 190.961,A -164.408,B 90.000,C 0.000} C_DIS
LIN {X 279.337,Y 77.914,Z 190.734,A -164.415,B 90.000,C 0.000} C_DIS
LIN {X 279.451,Y 77.505,Z 189.468,A -164.499,B 90.000,C 0.000} C_DIS
LIN {X 279.466,Y 77.453,Z 189.425,A -164.510,B 90.000,C 0.000} C_DIS
LIN {X 279.475,Y 77.420,Z 189.311,A -164.516,B 90.000,C 0.000} C_DIS
LIN {X 279.477,Y 77.411,Z 189.198,A -164.518,B 90.000,C 0.000} C_DIS
LIN {X 279.587,Y 77.015,Z 188.003,A -164.599,B 90.000,C 0.000} C_DIS
LIN {X 279.593,Y 76.993,Z 187.889,A -164.604,B 90.000,C 0.000} C_DIS
LIN {X 279.611,Y 76.926,Z 187.664,A -164.617,B 90.000,C 0.000} C_DIS
LIN {X 279.615,Y 76.910,Z 187.536,A -164.621,B 90.000,C 0.000} C_DIS
LIN {X 279.736,Y 76.472,Z 185.935,A -164.711,B 90.000,C 0.000} C_DIS
LIN {X 279.759,Y 76.387,Z 185.788,A -164.728,B 90.000,C 0.000} C_DIS
LIN {X 279.785,Y 76.291,Z 185.329,A -164.748,B 90.000,C 0.000} C_DIS
LIN {X 279.796,Y 76.249,Z 185.215,A -164.756,B 90.000,C 0.000} C_DIS
LIN {X 279.806,Y 76.215,Z 185.177,A -164.763,B 90.000,C 0.000} C_DIS
LIN {X 279.820,Y 76.162,Z 184.903,A -164.774,B 90.000,C 0.000} C_DIS
LIN {X 279.836,Y 76.103,Z 184.703,A -164.786,B 90.000,C 0.000} C_DIS
LIN {X 279.840,Y 76.089,Z 184.589,A -164.789,B 90.000,C 0.000} C_DIS
LIN {X 279.860,Y 76.017,Z 184.475,A -164.804,B 90.000,C 0.000} C_DIS
LIN {X 279.841,Y 76.084,Z 184.360,A -164.790,B 90.000,C 0.000} C_DIS
LIN {X 279.390,Y 77.724,Z 185.272,A -164.454,B 90.000,C 0.000} C_DIS
LIN {X 278.769,Y 79.925,Z 186.281,A -164.002,B 90.000,C 0.000} C_DIS
LIN {X 278.105,Y 82.197,Z 187.087,A -163.534,B 90.000,C 0.000} C_DIS
LIN {X 277.411,Y 84.512,Z 187.724,A -163.057,B 90.000,C 0.000} C_DIS
LIN {X 276.686,Y 86.862,Z 188.173,A -162.571,B 90.000,C 0.000} C_DIS
LIN {X 275.928,Y 89.236,Z 188.379,A -162.079,B 90.000,C 0.000} C_DIS
LIN {X 275.561,Y 90.365,Z 188.401,A -161.844,B 90.000,C 0.000} C_DIS
LIN {X 274.772,Y 92.736,Z 188.338,A -161.350,B 90.000,C 0.000} C_DIS
LIN {X 274.207,Y 94.397,Z 188.210,A -161.004,B 90.000,C 0.000} C_DIS
LIN {X 274.123,Y 94.640,Z 188.132,A -160.953,B 90.000,C 0.000} C_DIS
LIN {X 273.810,Y 95.541,Z 188.032,A -160.765,B 90.000,C 0.000} C_DIS
LIN {X 273.784,Y 95.616,Z 188.009,A -160.749,B 90.000,C 0.000} C_DIS
LIN {X 273.736,Y 95.754,Z 187.986,A -160.720,B 90.000,C 0.000} C_DIS
LIN {X 273.698,Y 95.861,Z 187.949,A -160.697,B 90.000,C 0.000} C_DIS
LIN {X 273.682,Y 95.908,Z 187.913,A -160.688,B 90.000,C 0.000} C_DIS
LIN {X 273.358,Y 96.828,Z 187.804,A -160.495,B 90.000,C 0.000} C_DIS
LIN {X 273.335,Y 96.891,Z 187.772,A -160.482,B 90.000,C 0.000} C_DIS
LIN {X 272.510,Y 99.175,Z 187.181,A -160.002,B 90.000,C 0.000} C_DIS
LIN {X 271.868,Y 100.934,Z 186.702,A -159.632,B 90.000,C 0.000} C_DIS
LIN {X 271.823,Y 101.055,Z 186.678,A -159.607,B 90.000,C 0.000} C_DIS
LIN {X 271.745,Y 101.265,Z 186.597,A -159.562,B 90.000,C 0.000} C_DIS
LIN {X 271.366,Y 102.278,Z 186.237,A -159.349,B 90.000,C 0.000} C_DIS
LIN {X 271.325,Y 102.384,Z 186.223,A -159.326,B 90.000,C 0.000} C_DIS
LIN {X 271.185,Y 102.757,Z 186.085,A -159.247,B 90.000,C 0.000} C_DIS
LIN {X 271.144,Y 102.863,Z 186.075,A -159.225,B 90.000,C 0.000} C_DIS
LIN {X 270.890,Y 103.530,Z 185.841,A -159.084,B 90.000,C 0.000} C_DIS
LIN {X 270.861,Y 103.607,Z 185.780,A -159.068,B 90.000,C 0.000} C_DIS
LIN {X 270.840,Y 103.661,Z 185.755,A -159.056,B 90.000,C 0.000} C_DIS
LIN {X 270.820,Y 103.714,Z 185.742,A -159.045,B 90.000,C 0.000} C_DIS
LIN {X 270.534,Y 104.457,Z 185.427,A -158.888,B 90.000,C 0.000} C_DIS
LIN {X 270.493,Y 104.563,Z 185.396,A -158.865,B 90.000,C 0.000} C_DIS
LIN {X 270.298,Y 105.068,Z 185.157,A -158.758,B 90.000,C 0.000} C_DIS
LIN {X 269.862,Y 106.181,Z 184.643,A -158.522,B 90.000,C 0.000} C_DIS
LIN {X 269.830,Y 106.263,Z 184.620,A -158.505,B 90.000,C 0.000} C_DIS
LIN {X 269.810,Y 106.312,Z 184.599,A -158.494,B 90.000,C 0.000} C_DIS
LIN {X 269.706,Y 106.577,Z 184.421,A -158.438,B 90.000,C 0.000} C_DIS
LIN {X 269.622,Y 106.789,Z 184.358,A -158.393,B 90.000,C 0.000} C_DIS
LIN {X 269.496,Y 107.106,Z 184.158,A -158.326,B 90.000,C 0.000} C_DIS
LIN {X 269.249,Y 107.727,Z 183.823,A -158.194,B 90.000,C 0.000} C_DIS
LIN {X 269.188,Y 107.879,Z 183.695,A -158.161,B 90.000,C 0.000} C_DIS
LIN {X 269.114,Y 108.063,Z 183.647,A -158.122,B 90.000,C 0.000} C_DIS
LIN {X 269.042,Y 108.243,Z 183.566,A -158.084,B 90.000,C 0.000} C_DIS
LIN {X 268.997,Y 108.353,Z 183.482,A -158.060,B 90.000,C 0.000} C_DIS
LIN {X 268.934,Y 108.509,Z 183.394,A -158.027,B 90.000,C 0.000} C_DIS
LIN {X 268.797,Y 108.849,Z 183.157,A -157.955,B 90.000,C 0.000} C_DIS
LIN {X 268.755,Y 108.954,Z 183.119,A -157.932,B 90.000,C 0.000} C_DIS
LIN {X 268.433,Y 109.744,Z 182.605,A -157.764,B 90.000,C 0.000} C_DIS
LIN {X 268.260,Y 110.166,Z 182.242,A -157.674,B 90.000,C 0.000} C_DIS
LIN {X 268.217,Y 110.271,Z 182.209,A -157.651,B 90.000,C 0.000} C_DIS
LIN {X 268.109,Y 110.534,Z 182.028,A -157.595,B 90.000,C 0.000} C_DIS
LIN {X 268.087,Y 110.587,Z 181.972,A -157.584,B 90.000,C 0.000} C_DIS
LIN {X 267.323,Y 112.421,Z 180.455,A -157.191,B 90.000,C 0.000} C_DIS
LIN {X 267.100,Y 112.950,Z 179.980,A -157.078,B 90.000,C 0.000} C_DIS
LIN {X 267.067,Y 113.028,Z 179.866,A -157.061,B 90.000,C 0.000} C_DIS
LIN {X 266.968,Y 113.262,Z 179.609,A -157.011,B 90.000,C 0.000} C_DIS
LIN {X 266.936,Y 113.336,Z 179.550,A -156.995,B 90.000,C 0.000} C_DIS
LIN {X 266.878,Y 113.473,Z 179.467,A -156.965,B 90.000,C 0.000} C_DIS
LIN {X 266.543,Y 114.258,Z 178.497,A -156.797,B 90.000,C 0.000} C_DIS
LIN {X 266.522,Y 114.306,Z 178.470,A -156.786,B 90.000,C 0.000} C_DIS
LIN {X 266.487,Y 114.388,Z 178.388,A -156.769,B 90.000,C 0.000} C_DIS
LIN {X 266.419,Y 114.546,Z 178.159,A -156.735,B 90.000,C 0.000} C_DIS
LIN {X 266.384,Y 114.627,Z 178.077,A -156.717,B 90.000,C 0.000} C_DIS
LIN {X 266.363,Y 114.676,Z 178.058,A -156.707,B 90.000,C 0.000} C_DIS
LIN {X 266.273,Y 114.885,Z 177.667,A -156.662,B 90.000,C 0.000} C_DIS
LIN {X 266.206,Y 115.042,Z 177.505,A -156.628,B 90.000,C 0.000} C_DIS
LIN {X 266.002,Y 115.512,Z 176.825,A -156.527,B 90.000,C 0.000} C_DIS
LIN {X 265.705,Y 116.194,Z 175.599,A -156.380,B 90.000,C 0.000} C_DIS
LIN {X 265.388,Y 116.915,Z 174.032,A -156.224,B 90.000,C 0.000} C_DIS
LIN {X 265.353,Y 116.995,Z 173.906,A -156.207,B 90.000,C 0.000} C_DIS
LIN {X 265.071,Y 117.632,Z 171.506,A -156.069,B 90.000,C 0.000} C_DIS
LIN {X 264.853,Y 118.123,Z 169.064,A -155.963,B 90.000,C 0.000} C_DIS
LIN {X 264.624,Y 118.634,Z 166.628,A -155.853,B 90.000,C 0.000} C_DIS
LIN {X 264.387,Y 119.161,Z 164.196,A -155.739,B 90.000,C 0.000} C_DIS
LIN {X 264.093,Y 119.811,Z 161.800,A -155.598,B 90.000,C 0.000} C_DIS
LIN {X 263.953,Y 120.120,Z 160.960,A -155.531,B 90.000,C 0.000} C_DIS
LIN {X 263.892,Y 120.255,Z 160.730,A -155.501,B 90.000,C 0.000} C_DIS
LIN {X 263.892,Y 120.255,Z 160.730,A -155.501,B 90.000,C 0.000} C_DIS
LIN {X 263.840,Y 120.368,Z 160.703,A -155.477,B 90.000,C 0.000} C_DIS
LIN {X 263.809,Y 120.436,Z 160.863,A -155.462,B 90.000,C 0.000} C_DIS
LIN {X 263.759,Y 120.546,Z 161.794,A -155.438,B 90.000,C 0.000} C_DIS
LIN {X 263.743,Y 120.581,Z 161.895,A -155.431,B 90.000,C 0.000} C_DIS
LIN {X 263.602,Y 120.889,Z 164.348,A -155.364,B 90.000,C 0.000} C_DIS
LIN {X 261.784,Y 120.055,Z 164.348,A -155.364,B 90.000,C 0.000} C_DIS
WAIT SEC 0.1
RET=EKI_SetBool("oxy","torchState",FALSE)
RET = EKI_Send("oxy","torchState")
LIN {X 245.422,Y 112.552,Z 164.348,A -155.364,B 90.000,C 0.000} C_DIS
LIN {X 245.692,Y 111.961,Z 160.730,A -155.501,B 90.000,C 0.000} C_DIS
LIN {X 262.072,Y 119.426,Z 160.730,A -155.501,B 90.000,C 0.000} C_DIS
LIN {X 263.892,Y 120.255,Z 160.730,A -155.501,B 90.000,C 0.000} C_DIS
WAIT SEC 1
RET=EKI_SetBool("oxy","torchState",TRUE)
RET = EKI_Send("oxy","torchState")
LIN {X 263.892,Y 120.255,Z 160.730,A -155.501,B 90.000,C 0.000} C_DIS
LIN {X 262.072,Y 119.426,Z 160.730,A -155.501,B 90.000,C 0.000} C_DIS
WAIT SEC 0.1
RET=EKI_SetBool("oxy","torchState",FALSE)
RET = EKI_Send("oxy","torchState")
LIN {X 245.692,Y 111.961,Z 160.730,A -155.501,B 90.000,C 0.000} C_DIS
LIN {X 227.389,Y 145.583,Z 155.421,A -147.371,B 90.000,C 0.000} C_DIS
LIN {X 242.548,Y 155.288,Z 155.421,A -147.371,B 90.000,C 0.000} C_DIS
LIN {X 244.232,Y 156.367,Z 155.421,A -147.371,B 90.000,C 0.000} C_DIS
WAIT SEC 1
RET=EKI_SetBool("oxy","torchState",TRUE)
RET = EKI_Send("oxy","torchState")
LIN {X 244.165,Y 156.472,Z 155.428,A -147.346,B 90.000,C 0.000} C_DIS
LIN {X 244.087,Y 156.594,Z 155.392,A -147.318,B 90.000,C 0.000} C_DIS
LIN {X 244.064,Y 156.629,Z 155.338,A -147.309,B 90.000,C 0.000} C_DIS
LIN {X 244.002,Y 156.725,Z 155.304,A -147.287,B 90.000,C 0.000} C_DIS
LIN {X 243.941,Y 156.821,Z 155.289,A -147.264,B 90.000,C 0.000} C_DIS
LIN {X 243.648,Y 157.276,Z 155.059,A -147.158,B 90.000,C 0.000} C_DIS
LIN {X 243.600,Y 157.350,Z 155.034,A -147.140,B 90.000,C 0.000} C_DIS
LIN {X 243.571,Y 157.395,Z 155.006,A -147.130,B 90.000,C 0.000} C_DIS
LIN {X 243.548,Y 157.431,Z 154.956,A -147.121,B 90.000,C 0.000} C_DIS
LIN {X 242.914,Y 158.407,Z 154.548,A -146.891,B 90.000,C 0.000} C_DIS
LIN {X 242.858,Y 158.492,Z 154.487,A -146.871,B 90.000,C 0.000} C_DIS
LIN {X 242.827,Y 158.540,Z 154.462,A -146.860,B 90.000,C 0.000} C_DIS
LIN {X 242.796,Y 158.588,Z 154.449,A -146.849,B 90.000,C 0.000} C_DIS
LIN {X 242.078,Y 159.682,Z 153.779,A -146.590,B 90.000,C 0.000} C_DIS
LIN {X 241.883,Y 159.977,Z 153.637,A -146.520,B 90.000,C 0.000} C_DIS
LIN {X 241.827,Y 160.061,Z 153.580,A -146.500,B 90.000,C 0.000} C_DIS
LIN {X 241.804,Y 160.097,Z 153.538,A -146.492,B 90.000,C 0.000} C_DIS
LIN {X 240.944,Y 161.387,Z 152.608,A -146.185,B 90.000,C 0.000} C_DIS
LIN {X 240.881,Y 161.482,Z 152.560,A -146.163,B 90.000,C 0.000} C_DIS
LIN {X 240.767,Y 161.652,Z 152.401,A -146.122,B 90.000,C 0.000} C_DIS
LIN {X 240.564,Y 161.954,Z 152.222,A -146.050,B 90.000,C 0.000} C_DIS
LIN {X 240.505,Y 162.041,Z 152.133,A -146.030,B 90.000,C 0.000} C_DIS
LIN {X 239.798,Y 163.086,Z 151.182,A -145.780,B 90.000,C 0.000} C_DIS
LIN {X 239.688,Y 163.247,Z 151.064,A -145.742,B 90.000,C 0.000} C_DIS
LIN {X 239.634,Y 163.327,Z 150.963,A -145.723,B 90.000,C 0.000} C_DIS
LIN {X 238.579,Y 164.864,Z 149.298,A -145.355,B 90.000,C 0.000} C_DIS
LIN {X 238.155,Y 165.476,Z 148.523,A -145.207,B 90.000,C 0.000} C_DIS
LIN {X 238.056,Y 165.618,Z 148.389,A -145.173,B 90.000,C 0.000} C_DIS
LIN {X 237.667,Y 166.176,Z 147.563,A -145.039,B 90.000,C 0.000} C_DIS
LIN {X 237.586,Y 166.291,Z 147.442,A -145.011,B 90.000,C 0.000} C_DIS
LIN {X 237.276,Y 166.734,Z 146.776,A -144.904,B 90.000,C 0.000} C_DIS
LIN {X 237.217,Y 166.817,Z 146.596,A -144.884,B 90.000,C 0.000} C_DIS
LIN {X 237.004,Y 167.119,Z 146.118,A -144.811,B 90.000,C 0.000} C_DIS
LIN {X 236.947,Y 167.201,Z 145.955,A -144.791,B 90.000,C 0.000} C_DIS
LIN {X 236.849,Y 167.340,Z 145.760,A -144.758,B 90.000,C 0.000} C_DIS
LIN {X 236.717,Y 167.526,Z 145.350,A -144.713,B 90.000,C 0.000} C_DIS
LIN {X 236.668,Y 167.596,Z 145.274,A -144.696,B 90.000,C 0.000} C_DIS
LIN {X 236.619,Y 167.665,Z 145.158,A -144.679,B 90.000,C 0.000} C_DIS
LIN {X 236.572,Y 167.732,Z 145.011,A -144.663,B 90.000,C 0.000} C_DIS
LIN {X 235.838,Y 168.762,Z 142.855,A -144.413,B 90.000,C 0.000} C_DIS
LIN {X 235.212,Y 169.633,Z 140.597,A -144.201,B 90.000,C 0.000} C_DIS
LIN {X 234.695,Y 170.347,Z 138.257,A -144.027,B 90.000,C 0.000} C_DIS
LIN {X 234.273,Y 170.927,Z 135.863,A -143.885,B 90.000,C 0.000} C_DIS
LIN {X 233.951,Y 171.368,Z 133.423,A -143.777,B 90.000,C 0.000} C_DIS
LIN {X 233.717,Y 171.687,Z 130.955,A -143.699,B 90.000,C 0.000} C_DIS
LIN {X 233.553,Y 171.909,Z 128.470,A -143.645,B 90.000,C 0.000} C_DIS
LIN {X 233.497,Y 171.986,Z 125.972,A -143.626,B 90.000,C 0.000} C_DIS
LIN {X 233.488,Y 171.998,Z 123.472,A -143.623,B 90.000,C 0.000} C_DIS
LIN {X 233.536,Y 171.933,Z 120.973,A -143.639,B 90.000,C 0.000} C_DIS
LIN {X 233.595,Y 171.853,Z 119.400,A -143.659,B 90.000,C 0.000} C_DIS
LIN {X 233.641,Y 171.791,Z 119.030,A -143.674,B 90.000,C 0.000} C_DIS
LIN {X 233.827,Y 171.537,Z 116.550,A -143.736,B 90.000,C 0.000} C_DIS
LIN {X 233.837,Y 171.523,Z 116.412,A -143.739,B 90.000,C 0.000} C_DIS
LIN {X 233.858,Y 171.494,Z 116.343,A -143.746,B 90.000,C 0.000} C_DIS
LIN {X 233.879,Y 171.467,Z 116.240,A -143.753,B 90.000,C 0.000} C_DIS
LIN {X 233.891,Y 171.450,Z 116.057,A -143.757,B 90.000,C 0.000} C_DIS
LIN {X 234.150,Y 171.096,Z 114.274,A -143.844,B 90.000,C 0.000} C_DIS
LIN {X 234.369,Y 170.796,Z 113.135,A -143.917,B 90.000,C 0.000} C_DIS
LIN {X 234.550,Y 170.548,Z 111.631,A -143.978,B 90.000,C 0.000} C_DIS
LIN {X 234.619,Y 170.452,Z 109.134,A -144.001,B 90.000,C 0.000} C_DIS
LIN {X 234.624,Y 170.445,Z 108.934,A -144.003,B 90.000,C 0.000} C_DIS
LIN {X 234.645,Y 170.416,Z 108.866,A -144.010,B 90.000,C 0.000} C_DIS
LIN {X 234.676,Y 170.374,Z 109.002,A -144.020,B 90.000,C 0.000} C_DIS
LIN {X 234.880,Y 170.092,Z 109.628,A -144.089,B 90.000,C 0.000} C_DIS
LIN {X 234.988,Y 169.943,Z 110.157,A -144.126,B 90.000,C 0.000} C_DIS
LIN {X 235.044,Y 169.866,Z 110.823,A -144.144,B 90.000,C 0.000} C_DIS
LIN {X 234.947,Y 170.000,Z 112.902,A -144.112,B 90.000,C 0.000} C_DIS
LIN {X 235.049,Y 169.859,Z 115.396,A -144.146,B 90.000,C 0.000} C_DIS
LIN {X 235.274,Y 169.547,Z 117.866,A -144.222,B 90.000,C 0.000} C_DIS
LIN {X 235.636,Y 169.043,Z 120.288,A -144.345,B 90.000,C 0.000} C_DIS
LIN {X 236.105,Y 168.388,Z 122.655,A -144.504,B 90.000,C 0.000} C_DIS
LIN {X 236.535,Y 167.784,Z 124.342,A -144.650,B 90.000,C 0.000} C_DIS
LIN {X 236.588,Y 167.708,Z 124.351,A -144.669,B 90.000,C 0.000} C_DIS
LIN {X 236.651,Y 167.619,Z 124.297,A -144.690,B 90.000,C 0.000} C_DIS
LIN {X 236.324,Y 168.080,Z 121.862,A -144.579,B 90.000,C 0.000} C_DIS
LIN {X 236.120,Y 168.367,Z 119.387,A -144.509,B 90.000,C 0.000} C_DIS
LIN {X 236.008,Y 168.523,Z 116.996,A -144.471,B 90.000,C 0.000} C_DIS
LIN {X 236.041,Y 168.478,Z 116.880,A -144.482,B 90.000,C 0.000} C_DIS
LIN {X 236.049,Y 168.466,Z 114.380,A -144.485,B 90.000,C 0.000} C_DIS
LIN {X 236.148,Y 168.327,Z 112.502,A -144.519,B 90.000,C 0.000} C_DIS
LIN {X 236.178,Y 168.285,Z 112.317,A -144.529,B 90.000,C 0.000} C_DIS
LIN {X 236.430,Y 167.932,Z 109.855,A -144.615,B 90.000,C 0.000} C_DIS
LIN {X 236.469,Y 167.876,Z 109.482,A -144.628,B 90.000,C 0.000} C_DIS
LIN {X 236.814,Y 167.389,Z 107.526,A -144.746,B 90.000,C 0.000} C_DIS
LIN {X 236.826,Y 167.372,Z 107.418,A -144.750,B 90.000,C 0.000} C_DIS
LIN {X 236.980,Y 167.154,Z 106.812,A -144.803,B 90.000,C 0.000} C_DIS
LIN {X 236.989,Y 167.141,Z 106.698,A -144.806,B 90.000,C 0.000} C_DIS
LIN {X 237.008,Y 167.115,Z 106.584,A -144.812,B 90.000,C 0.000} C_DIS
LIN {X 237.091,Y 166.997,Z 106.314,A -144.841,B 90.000,C 0.000} C_DIS
LIN {X 237.275,Y 166.736,Z 105.491,A -144.904,B 90.000,C 0.000} C_DIS
LIN {X 237.309,Y 166.686,Z 105.390,A -144.916,B 90.000,C 0.000} C_DIS
LIN {X 237.338,Y 166.645,Z 105.276,A -144.926,B 90.000,C 0.000} C_DIS
LIN {X 237.373,Y 166.596,Z 105.195,A -144.938,B 90.000,C 0.000} C_DIS
LIN {X 237.764,Y 166.037,Z 103.821,A -145.072,B 90.000,C 0.000} C_DIS
LIN {X 237.799,Y 165.987,Z 103.740,A -145.084,B 90.000,C 0.000} C_DIS
LIN {X 237.827,Y 165.946,Z 103.626,A -145.094,B 90.000,C 0.000} C_DIS
LIN {X 237.896,Y 165.847,Z 103.455,A -145.118,B 90.000,C 0.000} C_DIS
LIN {X 237.925,Y 165.807,Z 103.341,A -145.128,B 90.000,C 0.000} C_DIS
LIN {X 238.228,Y 165.370,Z 102.522,A -145.233,B 90.000,C 0.000} C_DIS
LIN {X 238.319,Y 165.240,Z 102.317,A -145.264,B 90.000,C 0.000} C_DIS
LIN {X 238.347,Y 165.199,Z 102.203,A -145.274,B 90.000,C 0.000} C_DIS
LIN {X 238.436,Y 165.070,Z 101.996,A -145.305,B 90.000,C 0.000} C_DIS
LIN {X 238.576,Y 164.868,Z 101.637,A -145.353,B 90.000,C 0.000} C_DIS
LIN {X 238.632,Y 164.787,Z 101.544,A -145.373,B 90.000,C 0.000} C_DIS
LIN {X 239.054,Y 164.174,Z 100.572,A -145.520,B 90.000,C 0.000} C_DIS
LIN {X 239.076,Y 164.142,Z 100.497,A -145.528,B 90.000,C 0.000} C_DIS
LIN {X 240.049,Y 162.716,Z 98.689,A -145.869,B 90.000,C 0.000} C_DIS
LIN {X 240.248,Y 162.422,Z 98.334,A -145.939,B 90.000,C 0.000} C_DIS
LIN {X 240.263,Y 162.400,Z 98.282,A -145.944,B 90.000,C 0.000} C_DIS
LIN {X 240.359,Y 162.258,Z 98.113,A -145.978,B 90.000,C 0.000} C_DIS
LIN {X 240.411,Y 162.181,Z 97.989,A -145.996,B 90.000,C 0.000} C_DIS
LIN {X 240.923,Y 161.419,Z 97.024,A -146.178,B 90.000,C 0.000} C_DIS
LIN {X 241.030,Y 161.259,Z 96.857,A -146.216,B 90.000,C 0.000} C_DIS
LIN {X 241.387,Y 160.725,Z 96.063,A -146.343,B 90.000,C 0.000} C_DIS
LIN {X 241.441,Y 160.643,Z 95.967,A -146.362,B 90.000,C 0.000} C_DIS
LIN {X 241.491,Y 160.568,Z 95.811,A -146.380,B 90.000,C 0.000} C_DIS
LIN {X 241.802,Y 160.099,Z 95.158,A -146.491,B 90.000,C 0.000} C_DIS
LIN {X 241.827,Y 160.061,Z 95.063,A -146.500,B 90.000,C 0.000} C_DIS
LIN {X 242.285,Y 159.367,Z 93.884,A -146.664,B 90.000,C 0.000} C_DIS
LIN {X 242.334,Y 159.294,Z 93.733,A -146.682,B 90.000,C 0.000} C_DIS
LIN {X 242.367,Y 159.242,Z 93.588,A -146.694,B 90.000,C 0.000} C_DIS
LIN {X 242.386,Y 159.214,Z 93.555,A -146.701,B 90.000,C 0.000} C_DIS
LIN {X 242.455,Y 159.108,Z 93.385,A -146.726,B 90.000,C 0.000} C_DIS
LIN {X 242.483,Y 159.067,Z 93.271,A -146.735,B 90.000,C 0.000} C_DIS
LIN {X 242.516,Y 159.016,Z 93.194,A -146.747,B 90.000,C 0.000} C_DIS
LIN {X 242.640,Y 158.826,Z 92.778,A -146.792,B 90.000,C 0.000} C_DIS
LIN {X 242.673,Y 158.775,Z 92.702,A -146.804,B 90.000,C 0.000} C_DIS
LIN {X 242.698,Y 158.739,Z 92.588,A -146.813,B 90.000,C 0.000} C_DIS
LIN {X 242.827,Y 158.540,Z 92.222,A -146.860,B 90.000,C 0.000} C_DIS
LIN {X 243.115,Y 158.099,Z 91.289,A -146.964,B 90.000,C 0.000} C_DIS
LIN {X 243.121,Y 158.090,Z 91.218,A -146.966,B 90.000,C 0.000} C_DIS
LIN {X 243.255,Y 157.883,Z 90.654,A -147.015,B 90.000,C 0.000} C_DIS
LIN {X 243.530,Y 157.458,Z 89.649,A -147.115,B 90.000,C 0.000} C_DIS
LIN {X 243.535,Y 157.451,Z 89.549,A -147.116,B 90.000,C 0.000} C_DIS
LIN {X 243.667,Y 157.247,Z 89.004,A -147.164,B 90.000,C 0.000} C_DIS
LIN {X 243.695,Y 157.202,Z 88.776,A -147.175,B 90.000,C 0.000} C_DIS
LIN {X 243.857,Y 156.951,Z 88.085,A -147.234,B 90.000,C 0.000} C_DIS
LIN {X 243.874,Y 156.925,Z 87.866,A -147.240,B 90.000,C 0.000} C_DIS
LIN {X 244.002,Y 156.725,Z 87.152,A -147.287,B 90.000,C 0.000} C_DIS
LIN {X 244.035,Y 156.675,Z 87.069,A -147.299,B 90.000,C 0.000} C_DIS
LIN {X 244.090,Y 156.589,Z 86.856,A -147.319,B 90.000,C 0.000} C_DIS
LIN {X 244.415,Y 156.082,Z 84.430,A -147.438,B 90.000,C 0.000} C_DIS
LIN {X 244.508,Y 155.936,Z 83.596,A -147.472,B 90.000,C 0.000} C_DIS
LIN {X 244.526,Y 155.908,Z 83.542,A -147.479,B 90.000,C 0.000} C_DIS
LIN {X 244.546,Y 155.877,Z 83.428,A -147.486,B 90.000,C 0.000} C_DIS
LIN {X 244.563,Y 155.849,Z 83.143,A -147.493,B 90.000,C 0.000} C_DIS
LIN {X 244.583,Y 155.817,Z 83.029,A -147.500,B 90.000,C 0.000} C_DIS
LIN {X 244.603,Y 155.787,Z 82.980,A -147.507,B 90.000,C 0.000} C_DIS
LIN {X 244.660,Y 155.697,Z 82.000,A -147.528,B 90.000,C 0.000} C_DIS
LIN {X 244.678,Y 155.668,Z 81.948,A -147.535,B 90.000,C 0.000} C_DIS
LIN {X 244.697,Y 155.639,Z 81.865,A -147.542,B 90.000,C 0.000} C_DIS
LIN {X 244.836,Y 155.420,Z 79.379,A -147.593,B 90.000,C 0.000} C_DIS
LIN {X 244.881,Y 155.349,Z 76.880,A -147.610,B 90.000,C 0.000} C_DIS
LIN {X 244.852,Y 155.395,Z 74.381,A -147.599,B 90.000,C 0.000} C_DIS
LIN {X 244.813,Y 155.457,Z 72.883,A -147.584,B 90.000,C 0.000} C_DIS
LIN {X 244.825,Y 155.438,Z 72.798,A -147.589,B 90.000,C 0.000} C_DIS
LIN {X 244.857,Y 155.387,Z 72.916,A -147.601,B 90.000,C 0.000} C_DIS
LIN {X 244.904,Y 155.313,Z 73.230,A -147.618,B 90.000,C 0.000} C_DIS
LIN {X 245.372,Y 154.571,Z 75.571,A -147.791,B 90.000,C 0.000} C_DIS
LIN {X 245.762,Y 153.952,Z 77.961,A -147.936,B 90.000,C 0.000} C_DIS
LIN {X 246.099,Y 153.411,Z 80.379,A -148.062,B 90.000,C 0.000} C_DIS
LIN {X 246.381,Y 152.958,Z 82.821,A -148.167,B 90.000,C 0.000} C_DIS
LIN {X 246.544,Y 152.697,Z 85.302,A -148.228,B 90.000,C 0.000} C_DIS
LIN {X 246.584,Y 152.631,Z 87.801,A -148.243,B 90.000,C 0.000} C_DIS
LIN {X 246.523,Y 152.729,Z 90.085,A -148.220,B 90.000,C 0.000} C_DIS
LIN {X 246.312,Y 153.069,Z 92.552,A -148.141,B 90.000,C 0.000} C_DIS
LIN {X 246.007,Y 153.560,Z 94.537,A -148.027,B 90.000,C 0.000} C_DIS
LIN {X 245.978,Y 153.607,Z 94.579,A -148.016,B 90.000,C 0.000} C_DIS
LIN {X 245.960,Y 153.635,Z 94.693,A -148.010,B 90.000,C 0.000} C_DIS
LIN {X 245.951,Y 153.649,Z 94.807,A -148.006,B 90.000,C 0.000} C_DIS
LIN {X 245.815,Y 153.866,Z 95.433,A -147.956,B 90.000,C 0.000} C_DIS
LIN {X 245.773,Y 153.934,Z 95.589,A -147.940,B 90.000,C 0.000} C_DIS
LIN {X 245.679,Y 154.083,Z 96.199,A -147.905,B 90.000,C 0.000} C_DIS
LIN {X 245.647,Y 154.134,Z 96.286,A -147.893,B 90.000,C 0.000} C_DIS
LIN {X 245.634,Y 154.156,Z 96.343,A -147.888,B 90.000,C 0.000} C_DIS
LIN {X 245.627,Y 154.167,Z 96.400,A -147.886,B 90.000,C 0.000} C_DIS
LIN {X 245.526,Y 154.328,Z 96.849,A -147.848,B 90.000,C 0.000} C_DIS
LIN {X 245.507,Y 154.357,Z 96.906,A -147.841,B 90.000,C 0.000} C_DIS
LIN {X 245.402,Y 154.525,Z 97.325,A -147.802,B 90.000,C 0.000} C_DIS
LIN {X 245.380,Y 154.560,Z 97.367,A -147.794,B 90.000,C 0.000} C_DIS
LIN {X 245.287,Y 154.708,Z 97.652,A -147.760,B 90.000,C 0.000} C_DIS
LIN {X 245.254,Y 154.759,Z 97.879,A -147.747,B 90.000,C 0.000} C_DIS
LIN {X 245.141,Y 154.938,Z 98.197,A -147.706,B 90.000,C 0.000} C_DIS
LIN {X 244.951,Y 155.238,Z 98.946,A -147.635,B 90.000,C 0.000} C_DIS
LIN {X 244.824,Y 155.439,Z 99.302,A -147.589,B 90.000,C 0.000} C_DIS
LIN {X 244.801,Y 155.476,Z 99.416,A -147.580,B 90.000,C 0.000} C_DIS
LIN {X 244.768,Y 155.527,Z 99.497,A -147.568,B 90.000,C 0.000} C_DIS
LIN {X 244.728,Y 155.590,Z 99.653,A -147.553,B 90.000,C 0.000} C_DIS
LIN {X 244.678,Y 155.668,Z 99.785,A -147.535,B 90.000,C 0.000} C_DIS
LIN {X 244.613,Y 155.770,Z 100.127,A -147.511,B 90.000,C 0.000} C_DIS
LIN {X 244.550,Y 155.870,Z 100.292,A -147.488,B 90.000,C 0.000} C_DIS
LIN {X 244.511,Y 155.930,Z 100.448,A -147.473,B 90.000,C 0.000} C_DIS
LIN {X 244.186,Y 156.439,Z 101.464,A -147.354,B 90.000,C 0.000} C_DIS
LIN {X 244.156,Y 156.486,Z 101.523,A -147.343,B 90.000,C 0.000} C_DIS
LIN {X 243.880,Y 156.916,Z 102.520,A -147.242,B 90.000,C 0.000} C_DIS
LIN {X 243.841,Y 156.976,Z 102.624,A -147.228,B 90.000,C 0.000} C_DIS
LIN {X 243.658,Y 157.259,Z 103.171,A -147.161,B 90.000,C 0.000} C_DIS
LIN {X 243.635,Y 157.296,Z 103.284,A -147.153,B 90.000,C 0.000} C_DIS
LIN {X 243.602,Y 157.347,Z 103.366,A -147.141,B 90.000,C 0.000} C_DIS
LIN {X 243.231,Y 157.920,Z 104.761,A -147.006,B 90.000,C 0.000} C_DIS
LIN {X 243.198,Y 157.971,Z 104.821,A -146.994,B 90.000,C 0.000} C_DIS
LIN {X 243.174,Y 158.008,Z 104.934,A -146.985,B 90.000,C 0.000} C_DIS
LIN {X 243.077,Y 158.157,Z 105.219,A -146.950,B 90.000,C 0.000} C_DIS
LIN {X 243.048,Y 158.201,Z 105.446,A -146.940,B 90.000,C 0.000} C_DIS
LIN {X 242.912,Y 158.410,Z 105.902,A -146.890,B 90.000,C 0.000} C_DIS
LIN {X 242.890,Y 158.444,Z 106.129,A -146.882,B 90.000,C 0.000} C_DIS
LIN {X 242.798,Y 158.584,Z 106.414,A -146.849,B 90.000,C 0.000} C_DIS
LIN {X 242.787,Y 158.601,Z 106.528,A -146.845,B 90.000,C 0.000} C_DIS
LIN {X 242.745,Y 158.666,Z 106.727,A -146.830,B 90.000,C 0.000} C_DIS
LIN {X 242.739,Y 158.675,Z 106.812,A -146.828,B 90.000,C 0.000} C_DIS
LIN {X 242.574,Y 158.927,Z 107.585,A -146.768,B 90.000,C 0.000} C_DIS
LIN {X 242.568,Y 158.936,Z 107.685,A -146.766,B 90.000,C 0.000} C_DIS
LIN {X 242.554,Y 158.958,Z 107.722,A -146.761,B 90.000,C 0.000} C_DIS
LIN {X 242.531,Y 158.992,Z 107.836,A -146.753,B 90.000,C 0.000} C_DIS
LIN {X 242.517,Y 159.013,Z 107.950,A -146.748,B 90.000,C 0.000} C_DIS
LIN {X 242.475,Y 159.078,Z 108.106,A -146.733,B 90.000,C 0.000} C_DIS
LIN {X 242.375,Y 159.230,Z 109.031,A -146.697,B 90.000,C 0.000} C_DIS
LIN {X 242.357,Y 159.258,Z 109.099,A -146.690,B 90.000,C 0.000} C_DIS
LIN {X 242.287,Y 159.364,Z 109.600,A -146.665,B 90.000,C 0.000} C_DIS
LIN {X 242.267,Y 159.395,Z 109.855,A -146.658,B 90.000,C 0.000} C_DIS
LIN {X 242.250,Y 159.421,Z 109.941,A -146.652,B 90.000,C 0.000} C_DIS
LIN {X 242.056,Y 159.714,Z 112.203,A -146.582,B 90.000,C 0.000} C_DIS
LIN {X 241.940,Y 159.891,Z 114.308,A -146.540,B 90.000,C 0.000} C_DIS
LIN {X 241.900,Y 159.951,Z 114.678,A -146.526,B 90.000,C 0.000} C_DIS
LIN {X 241.794,Y 160.111,Z 117.170,A -146.488,B 90.000,C 0.000} C_DIS
LIN {X 241.720,Y 160.223,Z 119.667,A -146.462,B 90.000,C 0.000} C_DIS
LIN {X 241.702,Y 160.251,Z 122.166,A -146.455,B 90.000,C 0.000} C_DIS
LIN {X 241.710,Y 160.238,Z 124.666,A -146.458,B 90.000,C 0.000} C_DIS
LIN {X 241.749,Y 160.179,Z 127.165,A -146.472,B 90.000,C 0.000} C_DIS
LIN {X 241.778,Y 160.136,Z 128.164,A -146.482,B 90.000,C 0.000} C_DIS
LIN {X 241.763,Y 160.158,Z 128.516,A -146.477,B 90.000,C 0.000} C_DIS
LIN {X 241.733,Y 160.204,Z 128.554,A -146.466,B 90.000,C 0.000} C_DIS
LIN {X 241.694,Y 160.263,Z 128.534,A -146.452,B 90.000,C 0.000} C_DIS
LIN {X 241.487,Y 160.575,Z 128.381,A -146.378,B 90.000,C 0.000} C_DIS
LIN {X 240.887,Y 161.473,Z 128.430,A -146.165,B 90.000,C 0.000} C_DIS
LIN {X 240.737,Y 161.697,Z 128.494,A -146.112,B 90.000,C 0.000} C_DIS
LIN {X 240.613,Y 161.881,Z 129.689,A -146.068,B 90.000,C 0.000} C_DIS
LIN {X 240.594,Y 161.909,Z 129.741,A -146.061,B 90.000,C 0.000} C_DIS
LIN {X 240.574,Y 161.938,Z 129.823,A -146.054,B 90.000,C 0.000} C_DIS
LIN {X 240.486,Y 162.069,Z 131.055,A -146.023,B 90.000,C 0.000} C_DIS
LIN {X 240.478,Y 162.081,Z 131.107,A -146.020,B 90.000,C 0.000} C_DIS
LIN {X 240.425,Y 162.160,Z 131.832,A -146.001,B 90.000,C 0.000} C_DIS
LIN {X 240.403,Y 162.193,Z 131.960,A -145.994,B 90.000,C 0.000} C_DIS
LIN {X 240.362,Y 162.254,Z 132.742,A -145.979,B 90.000,C 0.000} C_DIS
LIN {X 240.341,Y 162.284,Z 132.927,A -145.972,B 90.000,C 0.000} C_DIS
LIN {X 240.238,Y 162.437,Z 135.349,A -145.935,B 90.000,C 0.000} C_DIS
LIN {X 240.265,Y 162.397,Z 137.848,A -145.945,B 90.000,C 0.000} C_DIS
LIN {X 240.289,Y 162.361,Z 138.549,A -145.954,B 90.000,C 0.000} C_DIS
LIN {X 240.283,Y 162.370,Z 138.617,A -145.951,B 90.000,C 0.000} C_DIS
LIN {X 240.313,Y 162.327,Z 139.526,A -145.962,B 90.000,C 0.000} C_DIS
LIN {X 240.516,Y 162.024,Z 142.000,A -146.034,B 90.000,C 0.000} C_DIS
LIN {X 240.844,Y 161.537,Z 144.429,A -146.150,B 90.000,C 0.000} C_DIS
LIN {X 241.257,Y 160.919,Z 146.817,A -146.297,B 90.000,C 0.000} C_DIS
LIN {X 241.809,Y 160.088,Z 149.109,A -146.494,B 90.000,C 0.000} C_DIS
LIN {X 242.472,Y 159.082,Z 151.299,A -146.732,B 90.000,C 0.000} C_DIS
LIN {X 242.640,Y 158.826,Z 151.723,A -146.792,B 90.000,C 0.000} C_DIS
LIN {X 242.765,Y 158.635,Z 152.138,A -146.837,B 90.000,C 0.000} C_DIS
LIN {X 242.808,Y 158.570,Z 152.215,A -146.853,B 90.000,C 0.000} C_DIS
LIN {X 242.920,Y 158.398,Z 152.528,A -146.893,B 90.000,C 0.000} C_DIS
LIN {X 242.952,Y 158.349,Z 152.544,A -146.905,B 90.000,C 0.000} C_DIS
LIN {X 243.076,Y 158.159,Z 152.935,A -146.950,B 90.000,C 0.000} C_DIS
LIN {X 243.122,Y 158.087,Z 153.012,A -146.967,B 90.000,C 0.000} C_DIS
LIN {X 243.169,Y 158.016,Z 153.071,A -146.983,B 90.000,C 0.000} C_DIS
LIN {X 243.239,Y 157.908,Z 153.311,A -147.009,B 90.000,C 0.000} C_DIS
LIN {X 243.664,Y 157.251,Z 154.275,A -147.163,B 90.000,C 0.000} C_DIS
LIN {X 243.725,Y 157.156,Z 154.313,A -147.186,B 90.000,C 0.000} C_DIS
LIN {X 243.941,Y 156.821,Z 154.843,A -147.264,B 90.000,C 0.000} C_DIS
LIN {X 243.972,Y 156.773,Z 154.861,A -147.276,B 90.000,C 0.000} C_DIS
LIN {X 244.002,Y 156.725,Z 154.886,A -147.287,B 90.000,C 0.000} C_DIS
LIN {X 244.232,Y 156.367,Z 155.421,A -147.371,B 90.000,C 0.000} C_DIS
LIN {X 242.548,Y 155.288,Z 155.421,A -147.371,B 90.000,C 0.000} C_DIS
WAIT SEC 0.1
RET=EKI_SetBool("oxy","torchState",FALSE)
RET = EKI_Send("oxy","torchState")
LIN {X 227.389,Y 145.583,Z 155.421,A -147.371,B 90.000,C 0.000} C_DIS
LIN {X 218.323,Y 158.856,Z 156.275,A -143.960,B 90.000,C 0.000} C_DIS
LIN {X 232.877,Y 169.447,Z 156.275,A -143.960,B 90.000,C 0.000} C_DIS
LIN {X 234.495,Y 170.623,Z 156.275,A -143.960,B 90.000,C 0.000} C_DIS
WAIT SEC 1
RET=EKI_SetBool("oxy","torchState",TRUE)
RET = EKI_Send("oxy","torchState")
LIN {X 234.486,Y 170.635,Z 156.350,A -143.957,B 90.000,C 0.000} C_DIS
LIN {X 234.458,Y 170.674,Z 156.329,A -143.947,B 90.000,C 0.000} C_DIS
LIN {X 234.433,Y 170.708,Z 156.170,A -143.939,B 90.000,C 0.000} C_DIS
LIN {X 234.469,Y 170.658,Z 156.119,A -143.951,B 90.000,C 0.000} C_DIS
LIN {X 234.495,Y 170.623,Z 156.275,A -143.960,B 90.000,C 0.000} C_DIS
LIN {X 232.877,Y 169.447,Z 156.275,A -143.960,B 90.000,C 0.000} C_DIS
WAIT SEC 0.1
RET=EKI_SetBool("oxy","torchState",FALSE)
RET = EKI_Send("oxy","torchState")
LIN {X 218.323,Y 158.856,Z 156.275,A -143.960,B 90.000,C 0.000} C_DIS
LIN {X 216.852,Y 160.858,Z 137.268,A -143.432,B 90.000,C 0.000} C_DIS
LIN {X 231.308,Y 171.582,Z 137.268,A -143.432,B 90.000,C 0.000} C_DIS
LIN {X 232.915,Y 172.774,Z 137.268,A -143.432,B 90.000,C 0.000} C_DIS
WAIT SEC 1
RET=EKI_SetBool("oxy","torchState",TRUE)
RET = EKI_Send("oxy","torchState")
LIN {X 232.915,Y 172.774,Z 137.268,A -143.432,B 90.000,C 0.000} C_DIS
LIN {X 231.308,Y 171.582,Z 137.268,A -143.432,B 90.000,C 0.000} C_DIS
WAIT SEC 0.1
RET=EKI_SetBool("oxy","torchState",FALSE)
RET = EKI_Send("oxy","torchState")
LIN {X 216.851,Y 160.858,Z 137.268,A -143.432,B 90.000,C 0.000} C_DIS
LIN {X 242.202,Y 119.324,Z 205.072,A -153.772,B 90.000,C 0.000} C_DIS
LIN {X 258.349,Y 127.279,Z 205.072,A -153.772,B 90.000,C 0.000} C_DIS
LIN {X 260.143,Y 128.163,Z 205.072,A -153.772,B 90.000,C 0.000} C_DIS
WAIT SEC 1
RET=EKI_SetBool("oxy","torchState",TRUE)
RET = EKI_Send("oxy","torchState")
LIN {X 260.130,Y 128.189,Z 205.121,A -153.766,B 90.000,C 0.000} C_DIS
LIN {X 260.083,Y 128.284,Z 206.101,A -153.746,B 90.000,C 0.000} C_DIS
LIN {X 260.068,Y 128.315,Z 206.153,A -153.739,B 90.000,C 0.000} C_DIS
LIN {X 260.054,Y 128.342,Z 206.295,A -153.733,B 90.000,C 0.000} C_DIS
LIN {X 260.051,Y 128.350,Z 206.437,A -153.731,B 90.000,C 0.000} C_DIS
LIN {X 260.027,Y 128.397,Z 206.622,A -153.721,B 90.000,C 0.000} C_DIS
LIN {X 259.886,Y 128.683,Z 209.101,A -153.658,B 90.000,C 0.000} C_DIS
LIN {X 259.883,Y 128.690,Z 209.154,A -153.656,B 90.000,C 0.000} C_DIS
LIN {X 259.850,Y 128.756,Z 209.415,A -153.642,B 90.000,C 0.000} C_DIS
LIN {X 259.776,Y 128.906,Z 210.704,A -153.609,B 90.000,C 0.000} C_DIS
LIN {X 259.751,Y 128.955,Z 210.861,A -153.598,B 90.000,C 0.000} C_DIS
LIN {X 259.652,Y 129.154,Z 212.581,A -153.554,B 90.000,C 0.000} C_DIS
LIN {X 259.639,Y 129.180,Z 212.668,A -153.548,B 90.000,C 0.000} C_DIS
LIN {X 259.622,Y 129.214,Z 212.923,A -153.541,B 90.000,C 0.000} C_DIS
LIN {X 259.598,Y 129.263,Z 213.108,A -153.530,B 90.000,C 0.000} C_DIS
LIN {X 259.475,Y 129.510,Z 215.085,A -153.475,B 90.000,C 0.000} C_DIS
LIN {X 259.444,Y 129.571,Z 215.219,A -153.462,B 90.000,C 0.000} C_DIS
LIN {X 259.374,Y 129.711,Z 216.399,A -153.431,B 90.000,C 0.000} C_DIS
LIN {X 259.360,Y 129.740,Z 216.480,A -153.424,B 90.000,C 0.000} C_DIS
LIN {X 259.348,Y 129.763,Z 216.626,A -153.419,B 90.000,C 0.000} C_DIS
LIN {X 259.334,Y 129.792,Z 216.735,A -153.413,B 90.000,C 0.000} C_DIS
LIN {X 259.316,Y 129.827,Z 216.808,A -153.405,B 90.000,C 0.000} C_DIS
LIN {X 259.219,Y 130.020,Z 218.257,A -153.362,B 90.000,C 0.000} C_DIS
LIN {X 259.205,Y 130.049,Z 218.328,A -153.356,B 90.000,C 0.000} C_DIS
LIN {X 259.183,Y 130.094,Z 218.584,A -153.346,B 90.000,C 0.000} C_DIS
LIN {X 259.169,Y 130.122,Z 218.668,A -153.340,B 90.000,C 0.000} C_DIS
LIN {X 259.068,Y 130.322,Z 220.038,A -153.296,B 90.000,C 0.000} C_DIS
LIN {X 259.053,Y 130.352,Z 220.092,A -153.289,B 90.000,C 0.000} C_DIS
LIN {X 258.987,Y 130.483,Z 220.832,A -153.260,B 90.000,C 0.000} C_DIS
LIN {X 258.724,Y 131.004,Z 223.263,A -153.145,B 90.000,C 0.000} C_DIS
LIN {X 258.432,Y 131.579,Z 225.678,A -153.017,B 90.000,C 0.000} C_DIS
LIN {X 258.359,Y 131.722,Z 226.265,A -152.986,B 90.000,C 0.000} C_DIS
LIN {X 258.348,Y 131.743,Z 226.422,A -152.981,B 90.000,C 0.000} C_DIS
LIN {X 258.332,Y 131.775,Z 226.521,A -152.974,B 90.000,C 0.000} C_DIS
LIN {X 258.312,Y 131.813,Z 226.564,A -152.965,B 90.000,C 0.000} C_DIS
LIN {X 258.301,Y 131.836,Z 226.692,A -152.960,B 90.000,C 0.000} C_DIS
LIN {X 258.160,Y 132.112,Z 227.659,A -152.899,B 90.000,C 0.000} C_DIS
LIN {X 258.149,Y 132.133,Z 227.787,A -152.894,B 90.000,C 0.000} C_DIS
LIN {X 258.124,Y 132.182,Z 227.830,A -152.884,B 90.000,C 0.000} C_DIS
LIN {X 258.109,Y 132.212,Z 227.944,A -152.877,B 90.000,C 0.000} C_DIS
LIN {X 258.103,Y 132.223,Z 228.058,A -152.874,B 90.000,C 0.000} C_DIS
LIN {X 257.993,Y 132.438,Z 228.603,A -152.827,B 90.000,C 0.000} C_DIS
LIN {X 257.989,Y 132.445,Z 228.703,A -152.825,B 90.000,C 0.000} C_DIS
LIN {X 257.711,Y 132.985,Z 229.941,A -152.705,B 90.000,C 0.000} C_DIS
LIN {X 257.672,Y 133.061,Z 230.085,A -152.688,B 90.000,C 0.000} C_DIS
LIN {X 257.633,Y 133.137,Z 230.189,A -152.671,B 90.000,C 0.000} C_DIS
LIN {X 257.461,Y 133.468,Z 230.796,A -152.598,B 90.000,C 0.000} C_DIS
LIN {X 257.123,Y 134.118,Z 231.566,A -152.453,B 90.000,C 0.000} C_DIS
LIN {X 257.139,Y 134.088,Z 231.701,A -152.460,B 90.000,C 0.000} C_DIS
LIN {X 257.231,Y 133.911,Z 231.755,A -152.499,B 90.000,C 0.000} C_DIS
LIN {X 257.504,Y 133.386,Z 231.952,A -152.616,B 90.000,C 0.000} C_DIS
LIN {X 257.528,Y 133.339,Z 231.987,A -152.626,B 90.000,C 0.000} C_DIS
LIN {X 257.579,Y 133.241,Z 232.024,A -152.648,B 90.000,C 0.000} C_DIS
LIN {X 257.638,Y 133.127,Z 232.039,A -152.674,B 90.000,C 0.000} C_DIS
LIN {X 258.540,Y 131.366,Z 232.525,A -153.064,B 90.000,C 0.000} C_DIS
LIN {X 258.566,Y 131.314,Z 232.556,A -153.076,B 90.000,C 0.000} C_DIS
LIN {X 258.618,Y 131.213,Z 232.593,A -153.099,B 90.000,C 0.000} C_DIS
LIN {X 259.265,Y 129.930,Z 232.821,A -153.382,B 90.000,C 0.000} C_DIS
LIN {X 260.372,Y 127.689,Z 232.879,A -153.876,B 90.000,C 0.000} C_DIS
LIN {X 261.068,Y 126.268,Z 232.815,A -154.189,B 90.000,C 0.000} C_DIS
LIN {X 262.108,Y 124.094,Z 232.149,A -154.665,B 90.000,C 0.000} C_DIS
LIN {X 262.270,Y 123.752,Z 231.984,A -154.740,B 90.000,C 0.000} C_DIS
LIN {X 262.060,Y 124.195,Z 229.533,A -154.643,B 90.000,C 0.000} C_DIS
LIN {X 261.838,Y 124.662,Z 227.087,A -154.541,B 90.000,C 0.000} C_DIS
LIN {X 261.622,Y 125.115,Z 224.638,A -154.442,B 90.000,C 0.000} C_DIS
LIN {X 261.410,Y 125.559,Z 222.187,A -154.344,B 90.000,C 0.000} C_DIS
LIN {X 261.198,Y 125.999,Z 219.735,A -154.248,B 90.000,C 0.000} C_DIS
LIN {X 260.991,Y 126.427,Z 217.281,A -154.154,B 90.000,C 0.000} C_DIS
LIN {X 260.792,Y 126.836,Z 214.823,A -154.064,B 90.000,C 0.000} C_DIS
LIN {X 260.600,Y 127.230,Z 212.362,A -153.977,B 90.000,C 0.000} C_DIS
LIN {X 260.420,Y 127.599,Z 209.896,A -153.896,B 90.000,C 0.000} C_DIS
LIN {X 260.268,Y 127.909,Z 207.420,A -153.828,B 90.000,C 0.000} C_DIS
LIN {X 260.181,Y 128.085,Z 205.200,A -153.789,B 90.000,C 0.000} C_DIS
LIN {X 260.143,Y 128.163,Z 205.072,A -153.772,B 90.000,C 0.000} C_DIS
LIN {X 258.349,Y 127.279,Z 205.072,A -153.772,B 90.000,C 0.000} C_DIS
WAIT SEC 0.1
RET=EKI_SetBool("oxy","torchState",FALSE)
RET = EKI_Send("oxy","torchState")
LIN {X 242.202,Y 119.324,Z 205.072,A -153.772,B 90.000,C 0.000} C_DIS
LIN {X 236.763,Y 129.783,Z 57.796,A -151.270,B 90.000,C 0.000} C_DIS
LIN {X 252.547,Y 138.435,Z 57.796,A -151.270,B 90.000,C 0.000} C_DIS
LIN {X 254.300,Y 139.396,Z 57.796,A -151.270,B 90.000,C 0.000} C_DIS
WAIT SEC 1
RET=EKI_SetBool("oxy","torchState",TRUE)
RET = EKI_Send("oxy","torchState")
LIN {X 254.300,Y 139.396,Z 57.796,A -151.270,B 90.000,C 0.000} C_DIS
LIN {X 252.547,Y 138.435,Z 57.796,A -151.270,B 90.000,C 0.000} C_DIS
WAIT SEC 0.1
RET=EKI_SetBool("oxy","torchState",FALSE)
RET = EKI_Send("oxy","torchState")
LIN {X 236.762,Y 129.783,Z 57.796,A -151.270,B 90.000,C 0.000} C_DIS
LIN {X 243.327,Y 117.014,Z 46.344,A -154.318,B 90.000,C 0.000} C_DIS
LIN {X 259.548,Y 124.814,Z 46.344,A -154.318,B 90.000,C 0.000} C_DIS
LIN {X 261.351,Y 125.681,Z 46.344,A -154.318,B 90.000,C 0.000} C_DIS
WAIT SEC 1
RET=EKI_SetBool("oxy","torchState",TRUE)
RET = EKI_Send("oxy","torchState")
LIN {X 261.351,Y 125.681,Z 46.344,A -154.318,B 90.000,C 0.000} C_DIS
LIN {X 259.548,Y 124.815,Z 46.344,A -154.318,B 90.000,C 0.000} C_DIS
WAIT SEC 0.1
RET=EKI_SetBool("oxy","torchState",FALSE)
RET = EKI_Send("oxy","torchState")
LIN {X 216.290,Y 104.012,Z 46.344,A -154.318,B 90.000,C 0.000} C_DIS
PTP {A1 0.0,A2 -100.0,A3 150.0,A4 0.0,A5 -50.0,A6 0.0}


END
